C01826=1220.684,210.182,-57.626,-177.358,6.193,148.333
C01827=1220.680,210.431,-57.649,-177.356,6.195,148.332
C01828=1220.676,210.681,-57.674,-177.353,6.197,148.332
C01829=1220.671,210.929,-57.699,-177.350,6.199,148.332
C01830=1220.666,211.199,-57.725,-177.347,6.200,148.331
C01831=1220.661,211.469,-57.751,-177.345,6.202,148.331
C01832=1220.656,211.739,-57.778,-177.342,6.204,148.330
C01833=1220.651,212.011,-57.804,-177.339,6.206,148.330
C01834=1220.647,212.259,-57.829,-177.337,6.208,148.330
C01835=1220.642,212.508,-57.853,-177.334,6.209,148.329
C01836=1220.637,212.757,-57.877,-177.331,6.211,148.329
C01837=1220.633,213.006,-57.902,-177.329,6.213,148.329
C01838=1220.628,213.254,-57.926,-177.326,6.215,148.328
C01839=1220.623,213.503,-57.951,-177.323,6.217,148.328
C01840=1220.620,213.752,-57.975,-177.321,6.219,148.328
C01841=1220.614,214.001,-58.000,-177.318,6.220,148.328
C01842=1220.610,214.249,-58.024,-177.316,6.222,148.327
C01843=1220.606,214.498,-58.050,-177.313,6.224,148.327
C01844=1220.601,214.747,-58.074,-177.311,6.225,148.326
C01845=1220.596,214.995,-58.099,-177.308,6.227,148.326
C01846=1220.592,215.244,-58.123,-177.306,6.229,148.326
C01847=1220.587,215.493,-58.148,-177.303,6.231,148.325
C01848=1220.583,215.742,-58.172,-177.300,6.233,148.325
C01849=1220.578,215.991,-58.197,-177.298,6.234,148.325
C01850=1220.574,216.239,-58.221,-177.295,6.236,148.324
C01851=1220.569,216.487,-58.246,-177.292,6.238,148.324
C01852=1220.565,216.737,-58.271,-177.290,6.240,148.324
C01853=1220.560,216.985,-58.295,-177.287,6.242,148.323
C01854=1220.556,217.235,-58.321,-177.285,6.244,148.323
C01855=1220.551,217.483,-58.345,-177.282,6.246,148.323
C01856=1220.546,217.732,-58.369,-177.279,6.247,148.322
C01857=1220.543,217.980,-58.394,-177.277,6.250,148.322
C01858=1220.538,218.229,-58.419,-177.274,6.251,148.322
C01859=1220.532,218.478,-58.444,-177.272,6.252,148.322
C01860=1220.529,218.727,-58.468,-177.270,6.254,148.321
C01861=1220.524,218.975,-58.494,-177.267,6.256,148.321
C01862=1220.520,219.224,-58.518,-177.265,6.258,148.321
C01863=1220.515,219.473,-58.543,-177.262,6.260,148.320
C01864=1220.511,219.722,-58.568,-177.259,6.262,148.320
C01865=1220.506,219.970,-58.593,-177.257,6.264,148.320
C01866=1220.501,220.219,-58.617,-177.254,6.265,148.319
C01867=1220.497,220.468,-58.643,-177.251,6.267,148.319
C01868=1220.493,220.716,-58.667,-177.249,6.269,148.319
C01869=1220.488,220.965,-58.692,-177.246,6.271,148.318
C01870=1220.483,221.214,-58.717,-177.243,6.273,148.318
C01871=1220.479,221.463,-58.742,-177.241,6.275,148.318
C01872=1220.474,221.711,-58.767,-177.238,6.277,148.317
C01873=1220.470,221.960,-58.792,-177.236,6.279,148.317
C01874=1220.465,222.209,-58.817,-177.233,6.281,148.317
C01875=1220.461,222.457,-58.842,-177.231,6.282,148.317
C01876=1220.456,222.706,-58.867,-177.228,6.284,148.316
C01877=1220.451,222.955,-58.891,-177.226,6.286,148.316
C01878=1220.447,223.204,-58.917,-177.223,6.287,148.316
C01879=1220.443,223.452,-58.941,-177.221,6.289,148.315
C01880=1220.438,223.701,-58.967,-177.218,6.291,148.315
C01881=1220.433,223.950,-58.992,-177.216,6.293,148.315
C01882=1220.429,224.198,-59.017,-177.213,6.295,148.314
C01883=1220.425,224.447,-59.042,-177.210,6.297,148.314
C01884=1220.420,224.696,-59.067,-177.208,6.299,148.314
C01885=1220.415,224.944,-59.092,-177.206,6.301,148.314
C01886=1220.411,225.193,-59.118,-177.203,6.302,148.313
C01887=1220.406,225.442,-59.142,-177.200,6.304,148.313
C01888=1220.402,225.691,-59.168,-177.198,6.306,148.313
C01889=1220.398,225.939,-59.193,-177.195,6.308,148.312
C01890=1220.393,226.188,-59.218,-177.192,6.310,148.312
C01891=1220.389,226.437,-59.244,-177.190,6.312,148.312
C01892=1220.384,226.685,-59.268,-177.187,6.314,148.311
C01893=1220.379,226.934,-59.294,-177.185,6.316,148.311
C01894=1220.375,227.182,-59.320,-177.182,6.318,148.311
C01895=1220.370,227.432,-59.345,-177.180,6.319,148.311
C01896=1220.366,227.680,-59.369,-177.177,6.321,148.310
C01897=1220.362,227.928,-59.395,-177.174,6.323,148.310
C01898=1220.357,228.177,-59.420,-177.172,6.325,148.310
C01899=1220.352,228.426,-59.446,-177.169,6.327,148.309
C01900=1220.348,228.675,-59.471,-177.167,6.329,148.309
C01901=1220.343,228.923,-59.496,-177.164,6.331,148.309
C01902=1220.339,229.172,-59.522,-177.162,6.333,148.309
C01903=1220.334,229.420,-59.547,-177.159,6.335,148.308
C01904=1220.329,229.670,-59.572,-177.157,6.337,148.308
C01905=1220.325,229.919,-59.598,-177.154,6.338,148.308
C01906=1220.320,230.167,-59.623,-177.151,6.340,148.307
C01907=1220.316,230.415,-59.649,-177.149,6.342,148.307
C01908=1220.311,230.664,-59.674,-177.147,6.344,148.307
C01909=1220.307,230.913,-59.699,-177.144,6.346,148.306
C01910=1220.303,231.162,-59.725,-177.141,6.348,148.306
C01911=1220.298,231.410,-59.751,-177.139,6.350,148.306
C01912=1220.294,231.659,-59.776,-177.136,6.352,148.306
C01913=1220.289,231.907,-59.802,-177.133,6.354,148.305
C01914=1220.284,232.156,-59.827,-177.131,6.356,148.305
C01915=1220.280,232.405,-59.852,-177.129,6.358,148.305
C01916=1220.276,232.654,-59.878,-177.126,6.360,148.304
C01917=1220.271,232.902,-59.904,-177.123,6.361,148.304
C01918=1220.267,233.151,-59.929,-177.121,6.363,148.304
C01919=1220.262,233.400,-59.955,-177.118,6.365,148.303
C01920=1220.258,233.648,-59.980,-177.116,6.367,148.303
C01921=1220.253,233.896,-60.006,-177.113,6.369,148.303
C01922=1220.249,234.145,-60.032,-177.111,6.371,148.303
C01923=1220.244,234.393,-60.057,-177.108,6.373,148.302
C01924=1220.240,234.643,-60.082,-177.106,6.375,148.302
C01925=1220.236,234.892,-60.108,-177.103,6.377,148.302
C01926=1220.231,235.140,-60.134,-177.101,6.379,148.302
C01927=1220.227,235.388,-60.159,-177.098,6.381,148.301
C01928=1220.222,235.638,-60.186,-177.096,6.383,148.301
C01929=1220.217,235.886,-60.211,-177.093,6.384,148.301
C01930=1220.213,236.135,-60.237,-177.091,6.387,148.301
C01931=1220.208,236.383,-60.263,-177.088,6.388,148.300
C01932=1220.204,236.631,-60.289,-177.086,6.390,148.300
C01933=1220.200,236.880,-60.314,-177.083,6.392,148.300
C01934=1220.195,237.151,-60.342,-177.080,6.394,148.299
C01935=1220.190,237.423,-60.370,-177.077,6.397,148.299
C01936=1220.185,237.694,-60.399,-177.074,6.399,148.299
C01937=1220.180,237.966,-60.427,-177.072,6.400,148.298
C01938=1220.175,238.214,-60.453,-177.070,6.403,148.298
C01939=1220.171,238.463,-60.479,-177.067,6.405,148.298
C01940=1220.167,238.712,-60.504,-177.064,6.406,148.298
C01941=1220.162,238.961,-60.530,-177.062,6.408,148.297
C01942=1220.157,239.208,-60.557,-177.059,6.410,148.297
C01943=1220.153,239.457,-60.583,-177.057,6.412,148.297
C01944=1220.149,239.706,-60.608,-177.054,6.414,148.297
C01945=1220.144,239.955,-60.634,-177.051,6.417,148.296
C01946=1220.139,240.204,-60.660,-177.049,6.419,148.296
C01947=1220.135,240.452,-60.687,-177.047,6.421,148.296
C01948=1220.131,240.700,-60.712,-177.044,6.423,148.296
C01949=1220.126,240.949,-60.738,-177.041,6.425,148.295
C01950=1220.121,241.198,-60.764,-177.039,6.427,148.295
C01951=1220.118,241.446,-60.791,-177.036,6.428,148.295
C01952=1220.113,241.695,-60.816,-177.034,6.431,148.295
C01953=1220.108,241.944,-60.843,-177.031,6.432,148.294
C01954=1220.104,242.192,-60.868,-177.029,6.434,148.294
C01955=1220.100,242.441,-60.895,-177.026,6.436,148.294
C01956=1220.095,242.689,-60.921,-177.024,6.438,148.294
C01957=1220.090,242.939,-60.947,-177.021,6.440,148.293
C01958=1220.086,243.186,-60.973,-177.019,6.442,148.293
C01959=1220.081,243.435,-60.999,-177.016,6.444,148.293
C01960=1220.077,243.684,-61.025,-177.014,6.446,148.293
C01961=1220.073,243.932,-61.052,-177.011,6.448,148.292
C01962=1220.068,244.181,-61.078,-177.009,6.450,148.292
C01963=1220.064,244.429,-61.104,-177.006,6.453,148.292
C01964=1220.060,244.678,-61.130,-177.003,6.455,148.292
C01965=1220.054,244.927,-61.156,-177.001,6.457,148.291
C01966=1220.050,245.175,-61.183,-176.998,6.459,148.291
C01967=1220.045,245.424,-61.209,-176.996,6.461,148.291
C01968=1220.041,245.672,-61.235,-176.993,6.463,148.291
C01969=1220.037,245.921,-61.261,-176.991,6.464,148.290
C01970=1220.032,246.169,-61.288,-176.988,6.466,148.290
C01971=1220.028,246.418,-61.314,-176.986,6.469,148.290
C01972=1220.024,246.667,-61.341,-176.983,6.470,148.290
C01973=1220.019,246.916,-61.367,-176.981,6.472,148.289
C01974=1220.014,247.163,-61.393,-176.979,6.474,148.289
C01975=1220.010,247.412,-61.419,-176.976,6.476,148.289
C01976=1220.005,247.661,-61.446,-176.973,6.479,148.289
C01977=1220.001,247.909,-61.472,-176.970,6.481,148.288
C01978=1219.997,248.158,-61.498,-176.968,6.483,148.288
C01979=1219.992,248.407,-61.525,-176.966,6.485,148.288
C01980=1219.988,248.655,-61.551,-176.963,6.487,148.288
C01981=1219.984,248.903,-61.578,-176.961,6.489,148.287
C01982=1219.979,249.153,-61.605,-176.958,6.491,148.287
C01983=1219.975,249.401,-61.631,-176.956,6.493,148.287
C01984=1219.970,249.650,-61.657,-176.953,6.495,148.287
C01985=1219.966,249.898,-61.684,-176.951,6.497,148.286
C01986=1219.961,250.147,-61.711,-176.948,6.500,148.286
C01987=1219.957,250.395,-61.737,-176.945,6.501,148.286
C01988=1219.952,250.644,-61.764,-176.943,6.504,148.286
C01989=1219.948,250.892,-61.790,-176.940,6.506,148.285
C01990=1219.943,251.141,-61.817,-176.938,6.507,148.285
C01991=1219.939,251.390,-61.844,-176.935,6.510,148.285
C01992=1219.935,251.638,-61.870,-176.933,6.511,148.285
C01993=1219.930,251.886,-61.897,-176.930,6.513,148.284
C01994=1219.926,252.135,-61.923,-176.928,6.516,148.284
C01995=1219.921,252.384,-61.950,-176.925,6.518,148.284
C01996=1219.917,252.632,-61.977,-176.922,6.520,148.284
C01997=1219.913,252.880,-62.004,-176.920,6.522,148.284
C01998=1219.908,253.129,-62.030,-176.918,6.524,148.283
C01999=1219.904,253.378,-62.056,-176.915,6.526,148.283
C02000=1219.899,253.626,-62.083,-176.913,6.528,148.283
C02001=1219.894,253.875,-62.111,-176.910,6.530,148.283
C02002=1219.891,254.123,-62.137,-176.908,6.532,148.282
C02003=1219.886,254.372,-62.163,-176.905,6.535,148.282
C02004=1219.881,254.620,-62.190,-176.902,6.537,148.282
C02005=1219.877,254.869,-62.217,-176.900,6.539,148.282
C02006=1219.872,255.117,-62.244,-176.898,6.541,148.282
C02007=1219.868,255.366,-62.271,-176.895,6.543,148.281
C02008=1219.863,255.614,-62.298,-176.893,6.545,148.281
C02009=1219.859,255.862,-62.325,-176.890,6.547,148.281
C02010=1219.854,256.111,-62.352,-176.888,6.549,148.281
C02011=1219.850,256.359,-62.379,-176.885,6.552,148.281
C02012=1219.846,256.609,-62.405,-176.882,6.554,148.280
C02013=1219.841,256.857,-62.432,-176.880,6.556,148.280
C02014=1219.837,257.106,-62.459,-176.878,6.558,148.280
C02015=1219.832,257.354,-62.486,-176.875,6.560,148.280
C02016=1219.828,257.603,-62.513,-176.873,6.562,148.280
C02017=1219.824,257.851,-62.539,-176.870,6.565,148.279
C02018=1219.819,258.099,-62.567,-176.867,6.566,148.279
C02019=1219.814,258.348,-62.594,-176.865,6.569,148.279
C02020=1219.810,258.596,-62.621,-176.862,6.570,148.279
C02021=1219.806,258.846,-62.648,-176.860,6.572,148.278
C02022=1219.802,259.093,-62.675,-176.858,6.575,148.278
C02023=1219.797,259.342,-62.702,-176.855,6.576,148.278
C02024=1219.793,259.590,-62.729,-176.852,6.579,148.278
C02025=1219.788,259.839,-62.756,-176.850,6.581,148.278
C02026=1219.783,260.087,-62.783,-176.847,6.583,148.277
C02027=1219.779,260.336,-62.811,-176.845,6.585,148.277
C02028=1219.775,260.585,-62.837,-176.842,6.587,148.277
C02029=1219.771,260.833,-62.864,-176.840,6.589,148.277
C02030=1219.766,261.081,-62.892,-176.837,6.592,148.277
C02031=1219.762,261.329,-62.919,-176.835,6.594,148.276
C02032=1219.757,261.578,-62.946,-176.832,6.596,148.276
C02033=1219.752,261.826,-62.973,-176.830,6.598,148.276
C02034=1219.748,262.076,-63.001,-176.828,6.600,148.276
C02035=1219.744,262.324,-63.028,-176.824,6.603,148.275
C02036=1219.739,262.572,-63.056,-176.822,6.605,148.275
C02037=1219.735,262.820,-63.082,-176.820,6.607,148.275
C02038=1219.730,263.093,-63.112,-176.817,6.609,148.275
C02039=1219.725,263.366,-63.141,-176.814,6.612,148.275
C02040=1219.721,263.639,-63.172,-176.812,6.614,148.274
C02041=1219.716,263.911,-63.202,-176.809,6.617,148.274
C02042=1219.711,264.160,-63.229,-176.806,6.619,148.274
C02043=1219.707,264.408,-63.257,-176.804,6.621,148.274
C02044=1219.702,264.656,-63.284,-176.801,6.623,148.274
C02045=1219.698,264.905,-63.311,-176.799,6.626,148.273
C02046=1219.694,265.153,-63.339,-176.796,6.628,148.273
C02047=1219.689,265.402,-63.366,-176.794,6.630,148.273
C02048=1219.685,265.650,-63.393,-176.791,6.632,148.273
C02049=1219.681,265.899,-63.421,-176.789,6.634,148.273
C02050=1219.676,266.147,-63.448,-176.786,6.637,148.272
C02051=1219.672,266.395,-63.476,-176.784,6.639,148.272
C02052=1219.667,266.644,-63.503,-176.781,6.641,148.272
C02053=1219.663,266.893,-63.531,-176.779,6.643,148.272
C02054=1219.658,267.141,-63.559,-176.776,6.645,148.272
C02055=1219.654,267.390,-63.586,-176.774,6.648,148.272
C02056=1219.650,267.638,-63.614,-176.771,6.650,148.271
C02057=1219.645,267.887,-63.641,-176.769,6.652,148.271
C02058=1219.641,268.134,-63.669,-176.766,6.654,148.271
C02059=1219.636,268.383,-63.696,-176.763,6.656,148.271
C02060=1219.632,268.632,-63.724,-176.761,6.659,148.271
C02061=1219.628,268.880,-63.751,-176.759,6.660,148.270
C02062=1219.623,269.128,-63.779,-176.756,6.663,148.270
C02063=1219.619,269.377,-63.806,-176.753,6.665,148.270
C02064=1219.614,269.625,-63.835,-176.751,6.668,148.270
C02065=1219.610,269.874,-63.862,-176.749,6.669,148.270
C02066=1219.606,270.122,-63.890,-176.746,6.672,148.270
C02067=1219.601,270.371,-63.917,-176.744,6.674,148.269
C02068=1219.597,270.619,-63.945,-176.741,6.677,148.269
C02069=1219.593,270.867,-63.973,-176.738,6.678,148.269
C02070=1219.588,271.116,-64.001,-176.736,6.681,148.269
C02071=1219.583,271.364,-64.028,-176.734,6.683,148.269
C02072=1219.579,271.613,-64.056,-176.731,6.686,148.269
C02073=1219.575,271.861,-64.084,-176.729,6.688,148.269
C02074=1219.571,272.110,-64.112,-176.726,6.690,148.268
C02075=1219.566,272.358,-64.139,-176.724,6.692,148.268
C02076=1219.561,272.606,-64.167,-176.721,6.695,148.268
C02077=1219.558,272.855,-64.195,-176.719,6.697,148.268
C02078=1219.553,273.103,-64.222,-176.716,6.699,148.268
C02079=1219.548,273.352,-64.251,-176.714,6.701,148.267
C02080=1219.544,273.600,-64.279,-176.711,6.704,148.267
C02081=1219.540,273.848,-64.307,-176.709,6.706,148.267
C02082=1219.536,274.097,-64.334,-176.706,6.708,148.267
C02083=1219.531,274.345,-64.362,-176.704,6.710,148.267
C02084=1219.526,274.593,-64.390,-176.701,6.713,148.267
C02085=1219.523,274.842,-64.418,-176.699,6.715,148.266
C02086=1219.518,275.090,-64.445,-176.697,6.717,148.266
C02087=1219.513,275.339,-64.474,-176.694,6.719,148.266
C02088=1219.509,275.587,-64.502,-176.692,6.722,148.266
C02089=1219.505,275.836,-64.530,-176.689,6.724,148.266
C02090=1219.500,276.084,-64.559,-176.687,6.726,148.266
C02091=1219.496,276.332,-64.587,-176.684,6.729,148.265
C02092=1219.492,276.581,-64.614,-176.682,6.731,148.265
C02093=1219.487,276.829,-64.642,-176.679,6.733,148.265
C02094=1219.483,277.078,-64.670,-176.677,6.735,148.265
C02095=1219.479,277.326,-64.698,-176.674,6.738,148.265
C02096=1219.474,277.575,-64.727,-176.672,6.740,148.265
C02097=1219.470,277.822,-64.755,-176.669,6.742,148.265
C02098=1219.465,278.071,-64.783,-176.667,6.744,148.264
C02099=1219.461,278.319,-64.811,-176.664,6.747,148.264
C02100=1219.457,278.568,-64.839,-176.662,6.749,148.264
C02101=1219.452,278.816,-64.868,-176.659,6.751,148.264
C02102=1219.448,279.064,-64.896,-176.657,6.754,148.264
C02103=1219.443,279.313,-64.924,-176.654,6.756,148.264
C02104=1219.440,279.561,-64.952,-176.652,6.758,148.264
C02105=1219.435,279.809,-64.980,-176.650,6.760,148.263
C02106=1219.431,280.058,-65.009,-176.647,6.763,148.263
C02107=1219.426,280.306,-65.036,-176.645,6.765,148.263
C02108=1219.422,280.555,-65.065,-176.642,6.767,148.263
C02109=1219.418,280.803,-65.093,-176.639,6.770,148.263
C02110=1219.413,281.052,-65.122,-176.637,6.773,148.263
C02111=1219.409,281.299,-65.150,-176.635,6.774,148.262
C02112=1219.404,281.548,-65.178,-176.632,6.777,148.262
C02113=1219.400,281.797,-65.206,-176.630,6.780,148.262
C02114=1219.395,282.045,-65.235,-176.627,6.782,148.262
C02115=1219.392,282.293,-65.264,-176.625,6.784,148.262
C02116=1219.387,282.541,-65.292,-176.622,6.787,148.262
C02117=1219.383,282.790,-65.320,-176.620,6.789,148.262
C02118=1219.378,283.038,-65.349,-176.618,6.791,148.262
C02119=1219.374,283.287,-65.377,-176.615,6.794,148.262
C02120=1219.370,283.535,-65.405,-176.612,6.796,148.261
C02121=1219.365,283.783,-65.434,-176.610,6.798,148.261
C02122=1219.361,284.032,-65.463,-176.608,6.801,148.261
C02123=1219.356,284.280,-65.491,-176.605,6.803,148.261
C02124=1219.352,284.528,-65.519,-176.603,6.805,148.261
C02125=1219.347,284.777,-65.548,-176.600,6.808,148.261
C02126=1219.343,285.025,-65.577,-176.598,6.810,148.261
C02127=1219.339,285.273,-65.605,-176.595,6.812,148.261
C02128=1219.334,285.522,-65.633,-176.593,6.815,148.260
C02129=1219.331,285.770,-65.662,-176.590,6.817,148.260
C02130=1219.326,286.018,-65.691,-176.588,6.819,148.260
C02131=1219.321,286.267,-65.719,-176.585,6.822,148.260
C02132=1219.318,286.515,-65.748,-176.583,6.824,148.260
C02133=1219.313,286.763,-65.777,-176.581,6.827,148.260
C02134=1219.308,287.012,-65.805,-176.578,6.830,148.260
C02135=1219.305,287.260,-65.834,-176.575,6.831,148.259
C02136=1219.300,287.508,-65.863,-176.573,6.834,148.259
C02137=1219.295,287.757,-65.891,-176.571,6.837,148.259
C02138=1219.292,288.005,-65.920,-176.569,6.839,148.259
C02139=1219.287,288.253,-65.949,-176.566,6.841,148.259
C02140=1219.282,288.501,-65.978,-176.563,6.844,148.259
C02141=1219.278,288.750,-66.007,-176.561,6.846,148.259
C02142=1219.273,289.024,-66.038,-176.558,6.849,148.259
C02143=1219.268,289.299,-66.070,-176.556,6.851,148.259
C02144=1219.263,289.572,-66.102,-176.553,6.854,148.259
C02145=1219.258,289.846,-66.134,-176.550,6.857,148.258
C02146=1219.255,290.095,-66.162,-176.548,6.859,148.258
C02147=1219.251,290.343,-66.191,-176.546,6.861,148.258
C02148=1219.246,290.592,-66.220,-176.543,6.864,148.258
C02149=1219.241,290.839,-66.249,-176.541,6.866,148.258
C02150=1219.238,291.087,-66.278,-176.538,6.868,148.258
C02151=1219.233,291.336,-66.307,-176.536,6.871,148.258
C02152=1219.229,291.584,-66.336,-176.533,6.873,148.258
C02153=1219.224,291.833,-66.365,-176.531,6.875,148.258
C02154=1219.220,292.081,-66.394,-176.528,6.879,148.258
C02155=1219.215,292.330,-66.423,-176.526,6.881,148.257
C02156=1219.211,292.577,-66.451,-176.524,6.884,148.257
C02157=1219.207,292.825,-66.481,-176.521,6.886,148.257
C02158=1219.203,293.074,-66.509,-176.519,6.888,148.257
C02159=1219.199,293.322,-66.539,-176.516,6.891,148.257
C02160=1219.194,293.570,-66.568,-176.514,6.893,148.257
C02161=1219.189,293.819,-66.597,-176.511,6.895,148.257
C02162=1219.185,294.067,-66.626,-176.509,6.898,148.257
C02163=1219.182,294.315,-66.655,-176.507,6.900,148.257
C02164=1219.177,294.564,-66.684,-176.505,6.902,148.257
C02165=1219.172,294.812,-66.713,-176.502,6.906,148.257
C02166=1219.168,295.060,-66.742,-176.500,6.908,148.257
C02167=1219.164,295.308,-66.772,-176.497,6.910,148.256
C02168=1219.159,295.557,-66.801,-176.495,6.913,148.256
C02169=1219.155,295.805,-66.830,-176.492,6.915,148.256
C02170=1219.151,296.053,-66.859,-176.490,6.918,148.256
C02171=1219.146,296.301,-66.888,-176.488,6.920,148.256
C02172=1219.142,296.549,-66.918,-176.485,6.922,148.256
C02173=1219.138,296.798,-66.947,-176.482,6.925,148.256
C02174=1219.133,297.047,-66.976,-176.480,6.927,148.256
C02175=1219.129,297.295,-67.006,-176.478,6.930,148.256
C02176=1219.125,297.542,-67.035,-176.475,6.933,148.256
C02177=1219.120,297.791,-67.064,-176.473,6.935,148.256
C02178=1219.116,298.039,-67.094,-176.471,6.938,148.256
C02179=1219.112,298.288,-67.122,-176.468,6.940,148.255
C02180=1219.108,298.536,-67.152,-176.465,6.943,148.255
C02181=1219.103,298.784,-67.181,-176.463,6.945,148.255
C02182=1219.099,299.032,-67.210,-176.461,6.947,148.255
C02183=1219.094,299.280,-67.240,-176.458,6.950,148.255
C02184=1219.090,299.528,-67.269,-176.456,6.952,148.255
C02185=1219.086,299.777,-67.299,-176.454,6.955,148.255
C02186=1219.082,300.025,-67.328,-176.452,6.958,148.255
C02187=1219.078,300.273,-67.358,-176.449,6.960,148.255
C02188=1219.073,300.522,-67.387,-176.446,6.963,148.255
C02189=1219.069,300.770,-67.416,-176.444,6.965,148.255
C02190=1219.065,301.018,-67.446,-176.442,6.967,148.255
C02191=1219.060,301.266,-67.475,-176.439,6.970,148.255
C02192=1219.056,301.514,-67.504,-176.437,6.972,148.255
C02193=1219.052,301.762,-67.534,-176.435,6.975,148.255
C02194=1219.047,302.011,-67.564,-176.433,6.977,148.254
C02195=1219.043,302.259,-67.593,-176.430,6.981,148.254
C02196=1219.039,302.507,-67.623,-176.428,6.983,148.254
C02197=1219.034,302.756,-67.652,-176.426,6.985,148.254
C02198=1219.030,303.004,-67.682,-176.423,6.988,148.254
C02199=1219.026,303.251,-67.712,-176.421,6.990,148.254
C02200=1219.022,303.500,-67.741,-176.418,6.993,148.254
C02201=1219.017,303.748,-67.771,-176.416,6.995,148.254
C02202=1219.013,303.997,-67.801,-176.414,6.998,148.254
C02203=1219.009,304.245,-67.830,-176.411,7.000,148.254
C02204=1219.005,304.493,-67.860,-176.409,7.003,148.254
C02205=1219.001,304.741,-67.890,-176.406,7.006,148.254
C02206=1218.996,304.989,-67.920,-176.404,7.008,148.254
C02207=1218.992,305.238,-67.950,-176.402,7.010,148.254
C02208=1218.988,305.486,-67.979,-176.399,7.013,148.254
C02209=1218.983,305.734,-68.008,-176.397,7.015,148.254
C02210=1218.979,305.982,-68.039,-176.394,7.018,148.254
C02211=1218.974,306.230,-68.068,-176.392,7.021,148.254
C02212=1218.970,306.478,-68.098,-176.390,7.024,148.254
C02213=1218.966,306.726,-68.127,-176.387,7.026,148.254
C02214=1218.962,306.975,-68.158,-176.385,7.028,148.254
C02215=1218.957,307.223,-68.188,-176.383,7.031,148.254
C02216=1218.953,307.471,-68.217,-176.381,7.033,148.253
C02217=1218.949,307.719,-68.248,-176.378,7.036,148.253
C02218=1218.945,307.968,-68.277,-176.376,7.039,148.253
C02219=1218.940,308.216,-68.307,-176.374,7.041,148.254
C02220=1218.936,308.464,-68.338,-176.371,7.044,148.254
C02221=1218.932,308.712,-68.367,-176.369,7.046,148.254
C02222=1218.927,308.960,-68.397,-176.367,7.049,148.253
C02223=1218.923,309.208,-68.427,-176.365,7.052,148.253
C02224=1218.919,309.457,-68.457,-176.362,7.055,148.253
C02225=1218.915,309.704,-68.487,-176.360,7.057,148.253
C02226=1218.910,309.953,-68.517,-176.358,7.059,148.253
C02227=1218.906,310.200,-68.547,-176.355,7.062,148.253
C02228=1218.902,310.449,-68.577,-176.353,7.064,148.253
C02229=1218.897,310.697,-68.607,-176.350,7.067,148.253
C02230=1218.893,310.945,-68.637,-176.348,7.070,148.253
C02231=1218.888,311.194,-68.667,-176.345,7.073,148.253
C02232=1218.884,311.441,-68.697,-176.343,7.075,148.253
C02233=1218.881,311.690,-68.728,-176.341,7.077,148.253
C02234=1218.876,311.938,-68.758,-176.339,7.080,148.253
C02235=1218.872,312.186,-68.788,-176.337,7.083,148.253
C02236=1218.867,312.434,-68.818,-176.334,7.086,148.253
C02237=1218.863,312.682,-68.848,-176.332,7.088,148.253
C02238=1218.858,312.931,-68.878,-176.329,7.091,148.253
C02239=1218.854,313.178,-68.908,-176.327,7.093,148.253
C02240=1218.850,313.427,-68.938,-176.325,7.096,148.253
C02241=1218.846,313.674,-68.968,-176.323,7.098,148.253
C02242=1218.842,313.923,-69.000,-176.321,7.101,148.253
C02243=1218.837,314.171,-69.029,-176.318,7.104,148.253
C02244=1218.833,314.419,-69.060,-176.316,7.106,148.253
C02245=1218.829,314.667,-69.090,-176.313,7.109,148.253
C02246=1218.824,314.943,-69.124,-176.311,7.112,148.253
C02247=1218.820,315.219,-69.157,-176.309,7.115,148.253
C02248=1218.815,315.495,-69.191,-176.306,7.118,148.253
C02249=1218.810,315.771,-69.225,-176.303,7.121,148.253
C02250=1218.806,316.019,-69.255,-176.302,7.123,148.253
C02251=1218.801,316.267,-69.285,-176.299,7.126,148.253
C02252=1218.797,316.515,-69.315,-176.297,7.128,148.253
C02253=1218.793,316.763,-69.346,-176.294,7.131,148.253
C02254=1218.788,317.012,-69.377,-176.292,7.134,148.253
C02255=1218.785,317.260,-69.407,-176.290,7.137,148.253
C02256=1218.780,317.508,-69.438,-176.288,7.139,148.253
C02257=1218.776,317.755,-69.468,-176.285,7.142,148.253
C02258=1218.771,318.003,-69.498,-176.283,7.144,148.253
C02259=1218.767,318.253,-69.529,-176.280,7.148,148.253
C02260=1218.763,318.500,-69.559,-176.279,7.150,148.254
C02261=1218.759,318.748,-69.590,-176.277,7.152,148.253
C02262=1218.754,318.996,-69.621,-176.274,7.155,148.253
C02263=1218.751,319.245,-69.651,-176.272,7.158,148.253
C02264=1218.746,319.493,-69.682,-176.270,7.161,148.254
C02265=1218.742,319.740,-69.712,-176.268,7.163,148.254
C02266=1218.738,319.988,-69.743,-176.265,7.166,148.254
C02267=1218.734,320.237,-69.774,-176.263,7.168,148.254
C02268=1218.729,320.485,-69.803,-176.261,7.172,148.254
C02269=1218.725,320.733,-69.834,-176.259,7.174,148.254
C02270=1218.720,320.981,-69.865,-176.256,7.176,148.254
C02271=1218.716,321.230,-69.896,-176.254,7.180,148.254
C02272=1218.712,321.477,-69.926,-176.252,7.182,148.254
C02273=1218.708,321.725,-69.957,-176.249,7.185,148.254
C02274=1218.703,321.973,-69.988,-176.248,7.187,148.254
C02275=1218.700,322.222,-70.018,-176.245,7.190,148.254
C02276=1218.695,322.470,-70.049,-176.243,7.193,148.254
C02277=1218.691,322.717,-70.080,-176.240,7.196,148.254
C02278=1218.687,322.966,-70.111,-176.239,7.198,148.254
C02279=1218.683,323.214,-70.141,-176.237,7.200,148.254
C02280=1218.678,323.461,-70.173,-176.234,7.204,148.254
C02281=1218.674,323.710,-70.204,-176.232,7.206,148.254
C02282=1218.670,323.958,-70.234,-176.230,7.209,148.254
C02283=1218.665,324.206,-70.265,-176.228,7.211,148.254
C02284=1218.662,324.454,-70.296,-176.225,7.215,148.254
C02285=1218.657,324.702,-70.327,-176.223,7.217,148.254
C02286=1218.653,324.950,-70.357,-176.221,7.220,148.255
C02287=1218.649,325.199,-70.388,-176.219,7.222,148.255
C02288=1218.644,325.446,-70.420,-176.216,7.225,148.255
C02289=1218.640,325.694,-70.450,-176.215,7.228,148.255
C02290=1218.636,325.942,-70.481,-176.213,7.230,148.255
C02291=1218.632,326.190,-70.512,-176.210,7.233,148.255
C02292=1218.627,326.438,-70.543,-176.208,7.236,148.255
C02293=1218.624,326.686,-70.575,-176.206,7.239,148.255
C02294=1218.619,326.934,-70.605,-176.204,7.241,148.255
C02295=1218.615,327.183,-70.636,-176.201,7.244,148.255
C02296=1218.611,327.430,-70.667,-176.200,7.247,148.255
C02297=1218.606,327.678,-70.697,-176.197,7.250,148.255
C02298=1218.603,327.926,-70.729,-176.195,7.252,148.255
C02299=1218.598,328.174,-70.760,-176.193,7.255,148.255
C02300=1218.593,328.422,-70.791,-176.191,7.258,148.256
C02301=1218.590,328.670,-70.823,-176.189,7.260,148.256
C02302=1218.585,328.918,-70.853,-176.186,7.263,148.256
C02303=1218.581,329.167,-70.885,-176.185,7.266,148.256
C02304=1218.577,329.414,-70.916,-176.182,7.269,148.256
C02305=1218.573,329.663,-70.947,-176.180,7.271,148.256
C02306=1218.568,329.911,-70.978,-176.178,7.274,148.256
C02307=1218.564,330.158,-71.009,-176.176,7.277,148.256
C02308=1218.560,330.407,-71.041,-176.173,7.280,148.256
C02309=1218.556,330.654,-71.072,-176.172,7.282,148.256
C02310=1218.552,330.903,-71.103,-176.170,7.285,148.256
C02311=1218.547,331.151,-71.134,-176.167,7.288,148.256
C02312=1218.543,331.399,-71.166,-176.166,7.291,148.257
C02313=1218.539,331.647,-71.197,-176.163,7.294,148.257
C02314=1218.534,331.894,-71.228,-176.161,7.296,148.257
C02315=1218.530,332.143,-71.259,-176.159,7.299,148.257
C02316=1218.526,332.390,-71.291,-176.157,7.302,148.257
C02317=1218.522,332.639,-71.322,-176.155,7.305,148.257
C02318=1218.518,332.886,-71.353,-176.153,7.307,148.257
C02319=1218.514,333.135,-71.384,-176.150,7.310,148.257
C02320=1218.509,333.382,-71.416,-176.149,7.313,148.257
C02321=1218.505,333.631,-71.447,-176.147,7.315,148.258
C02322=1218.501,333.878,-71.478,-176.144,7.318,148.258
C02323=1218.497,334.127,-71.510,-176.143,7.321,148.258
C02324=1218.493,334.374,-71.541,-176.140,7.324,148.258
C02325=1218.488,334.623,-71.573,-176.138,7.327,148.258
C02326=1218.484,334.871,-71.604,-176.136,7.330,148.258
C02327=1218.480,335.119,-71.636,-176.134,7.332,148.258
C02328=1218.475,335.367,-71.667,-176.132,7.335,148.258
C02329=1218.472,335.615,-71.699,-176.130,7.338,148.258
C02330=1218.467,335.862,-71.730,-176.128,7.340,148.258
C02331=1218.463,336.111,-71.761,-176.126,7.344,148.259
C02332=1218.459,336.358,-71.793,-176.124,7.346,148.259
C02333=1218.455,336.606,-71.825,-176.122,7.349,148.259
C02334=1218.451,336.855,-71.856,-176.120,7.352,148.259
C02335=1218.446,337.102,-71.888,-176.118,7.355,148.259
C02336=1218.443,337.350,-71.920,-176.116,7.357,148.259
C02337=1218.438,337.598,-71.950,-176.114,7.360,148.259
C02338=1218.433,337.847,-71.983,-176.112,7.363,148.260
C02339=1218.429,338.094,-72.014,-176.110,7.365,148.260
C02340=1218.425,338.342,-72.046,-176.108,7.369,148.260
C02341=1218.421,338.591,-72.077,-176.106,7.371,148.260
C02342=1218.417,338.838,-72.109,-176.103,7.374,148.260
C02343=1218.413,339.086,-72.141,-176.102,7.377,148.260
C02344=1218.408,339.334,-72.173,-176.100,7.379,148.260
C02345=1218.405,339.582,-72.205,-176.098,7.383,148.261
C02346=1218.400,339.830,-72.235,-176.096,7.385,148.261
C02347=1218.396,340.078,-72.268,-176.093,7.388,148.261
C02348=1218.392,340.326,-72.300,-176.092,7.391,148.261
C02349=1218.388,340.573,-72.331,-176.090,7.394,148.261
C02350=1218.383,340.851,-72.367,-176.088,7.396,148.261
C02351=1218.378,341.129,-72.402,-176.085,7.400,148.261
C02352=1218.374,341.407,-72.438,-176.083,7.403,148.262
C02353=1218.369,341.685,-72.474,-176.081,7.406,148.262
C02354=1218.365,341.933,-72.506,-176.079,7.409,148.262
C02355=1218.361,342.181,-72.538,-176.077,7.412,148.262
C02356=1218.356,342.429,-72.570,-176.075,7.414,148.262
C02357=1218.352,342.677,-72.601,-176.073,7.418,148.262
C02358=1218.348,342.926,-72.633,-176.071,7.420,148.263
C02359=1218.343,343.173,-72.665,-176.070,7.423,148.263
C02360=1218.340,343.421,-72.697,-176.067,7.426,148.263
C02361=1218.335,343.669,-72.729,-176.066,7.429,148.263
C02362=1218.331,343.917,-72.761,-176.063,7.432,148.263
C02363=1218.327,344.165,-72.792,-176.061,7.434,148.263
C02364=1218.322,344.412,-72.825,-176.059,7.438,148.264
C02365=1218.318,344.660,-72.856,-176.058,7.440,148.264
C02366=1218.314,344.909,-72.889,-176.056,7.443,148.264
C02367=1218.311,345.156,-72.921,-176.054,7.446,148.264
C02368=1218.306,345.403,-72.953,-176.052,7.449,148.264
C02369=1218.302,345.652,-72.985,-176.050,7.452,148.265
C02370=1218.298,345.900,-73.017,-176.048,7.454,148.265
C02371=1218.293,346.147,-73.049,-176.047,7.457,148.265
C02372=1218.289,346.395,-73.081,-176.044,7.460,148.265
C02373=1218.285,346.644,-73.113,-176.042,7.463,148.265
C02374=1218.281,346.891,-73.145,-176.040,7.466,148.265
C02375=1218.276,347.140,-73.177,-176.039,7.468,148.266
C02376=1218.273,347.387,-73.210,-176.037,7.471,148.266
C02377=1218.268,347.635,-73.242,-176.035,7.474,148.266
C02378=1218.264,347.883,-73.274,-176.033,7.477,148.266
C02379=1218.260,348.131,-73.306,-176.031,7.480,148.266
C02380=1218.256,348.379,-73.338,-176.029,7.483,148.267
C02381=1218.251,348.627,-73.370,-176.028,7.485,148.267
C02382=1218.247,348.874,-73.403,-176.025,7.489,148.267
C02383=1218.243,349.122,-73.435,-176.024,7.491,148.267
C02384=1218.239,349.370,-73.467,-176.022,7.494,148.267
C02385=1218.234,349.618,-73.499,-176.020,7.497,148.268
C02386=1218.231,349.866,-73.532,-176.018,7.500,148.268
C02387=1218.226,350.114,-73.564,-176.017,7.503,148.268
C02388=1218.223,350.362,-73.596,-176.015,7.506,148.268
C02389=1218.219,350.610,-73.629,-176.013,7.508,148.269
C02390=1218.214,350.857,-73.661,-176.011,7.512,148.269
C02391=1218.210,351.105,-73.693,-176.009,7.514,148.269
C02392=1218.206,351.353,-73.726,-176.007,7.517,148.269
C02393=1218.202,351.601,-73.758,-176.006,7.520,148.269
C02394=1218.197,351.849,-73.790,-176.004,7.522,148.270
C02395=1218.193,352.096,-73.823,-176.002,7.526,148.270
C02396=1218.189,352.345,-73.855,-176.000,7.528,148.270
C02397=1218.185,352.593,-73.888,-175.999,7.531,148.270
C02398=1218.181,352.840,-73.920,-175.997,7.535,148.271
C02399=1218.177,353.089,-73.953,-175.995,7.537,148.271
C02400=1218.173,353.335,-73.985,-175.993,7.540,148.271
C02401=1218.168,353.584,-74.017,-175.991,7.543,148.271
C02402=1218.164,353.832,-74.050,-175.990,7.545,148.271
C02403=1218.160,354.079,-74.082,-175.988,7.549,148.272
C02404=1218.156,354.328,-74.115,-175.986,7.552,148.272
C02405=1218.151,354.575,-74.147,-175.985,7.554,148.272
C02406=1218.148,354.823,-74.179,-175.982,7.558,148.272
C02407=1218.143,355.071,-74.212,-175.981,7.560,148.273
C02408=1218.139,355.319,-74.245,-175.980,7.563,148.273
C02409=1218.135,355.567,-74.278,-175.977,7.566,148.273
C02410=1218.131,355.815,-74.310,-175.976,7.569,148.273
C02411=1218.127,356.062,-74.343,-175.974,7.571,148.274
C02412=1218.122,356.310,-74.375,-175.972,7.575,148.274
C02413=1218.119,356.558,-74.408,-175.971,7.577,148.274
C02414=1218.114,356.806,-74.440,-175.969,7.580,148.274
C02415=1218.110,357.054,-74.473,-175.967,7.583,148.275
C02416=1218.106,357.301,-74.506,-175.966,7.586,148.275
C02417=1218.102,357.549,-74.538,-175.964,7.589,148.275
C02418=1218.098,357.797,-74.571,-175.962,7.592,148.275
C02419=1218.094,358.045,-74.604,-175.961,7.595,148.276
C02420=1218.089,358.293,-74.637,-175.959,7.597,148.276
C02421=1218.085,358.540,-74.669,-175.957,7.601,148.276
C02422=1218.081,358.788,-74.702,-175.956,7.604,148.277
C02423=1218.077,359.036,-74.735,-175.954,7.606,148.277
C02424=1218.073,359.284,-74.768,-175.952,7.609,148.277
C02425=1218.069,359.532,-74.800,-175.951,7.612,148.277
C02426=1218.065,359.779,-74.833,-175.949,7.615,148.278
C02427=1218.061,360.027,-74.866,-175.948,7.618,148.278
C02428=1218.056,360.276,-74.899,-175.946,7.621,148.278
C02429=1218.052,360.523,-74.932,-175.944,7.623,148.278
C02430=1218.048,360.771,-74.965,-175.943,7.626,148.279
C02431=1218.045,361.018,-74.997,-175.941,7.630,148.279
C02432=1218.040,361.267,-75.030,-175.939,7.632,148.279
C02433=1218.036,361.515,-75.063,-175.938,7.635,148.280
C02434=1218.032,361.762,-75.096,-175.937,7.638,148.280
C02435=1218.028,362.010,-75.129,-175.934,7.641,148.280
C02436=1218.024,362.258,-75.163,-175.933,7.644,148.280
C02437=1218.019,362.505,-75.195,-175.932,7.646,148.281
C02438=1218.015,362.753,-75.227,-175.929,7.650,148.281
C02439=1218.011,363.001,-75.260,-175.928,7.653,148.281
C02440=1218.007,363.248,-75.293,-175.927,7.655,148.282
C02441=1218.003,363.496,-75.327,-175.925,7.658,148.282
C02442=1217.999,363.744,-75.360,-175.923,7.661,148.282
C02443=1217.994,363.992,-75.392,-175.922,7.664,148.283
C02444=1217.990,364.240,-75.425,-175.921,7.667,148.283
C02445=1217.986,364.488,-75.459,-175.919,7.670,148.283
C02446=1217.982,364.735,-75.492,-175.918,7.672,148.284
C02447=1217.978,364.983,-75.525,-175.916,7.676,148.284
C02448=1217.973,365.231,-75.558,-175.915,7.679,148.284
C02449=1217.970,365.478,-75.591,-175.913,7.681,148.284
C02450=1217.966,365.726,-75.624,-175.912,7.684,148.285
C02451=1217.962,365.974,-75.657,-175.910,7.687,148.285
C02452=1217.958,366.221,-75.690,-175.908,7.690,148.286
C02453=1217.954,366.470,-75.724,-175.907,7.693,148.286
C02454=1217.949,366.750,-75.760,-175.906,7.696,148.286
C02455=1217.944,367.030,-75.798,-175.904,7.699,148.287
C02456=1217.939,367.309,-75.836,-175.902,7.703,148.287
C02457=1217.934,367.590,-75.873,-175.901,7.705,148.287
C02458=1217.930,367.837,-75.906,-175.899,7.709,148.288
C02459=1217.927,368.086,-75.940,-175.898,7.712,148.288
C02460=1217.923,368.334,-75.973,-175.896,7.714,148.288
C02461=1217.918,368.581,-76.006,-175.895,7.717,148.289
C02462=1217.915,368.828,-76.040,-175.894,7.720,148.289
C02463=1217.910,369.076,-76.073,-175.892,7.723,148.289
C02464=1217.906,369.324,-76.106,-175.891,7.725,148.290
C02465=1217.902,369.572,-76.139,-175.889,7.729,148.290
C02466=1217.898,369.819,-76.172,-175.888,7.732,148.290
C02467=1217.894,370.067,-76.205,-175.887,7.734,148.291
C02468=1217.890,370.315,-76.239,-175.885,7.737,148.291
C02469=1217.886,370.562,-76.272,-175.884,7.740,148.292
C02470=1217.881,370.810,-76.305,-175.883,7.743,148.292
C02471=1217.877,371.058,-76.338,-175.881,7.745,148.292
C02472=1217.873,371.305,-76.373,-175.880,7.748,148.293
C02473=1217.869,371.554,-76.406,-175.879,7.751,148.293
C02474=1217.865,371.802,-76.439,-175.877,7.755,148.293
C02475=1217.861,372.049,-76.472,-175.876,7.758,148.294
C02476=1217.857,372.297,-76.506,-175.875,7.760,148.294
C02477=1217.853,372.545,-76.539,-175.873,7.763,148.294
C02478=1217.849,372.792,-76.573,-175.872,7.766,148.295
C02479=1217.845,373.040,-76.606,-175.871,7.769,148.295
C02480=1217.840,373.288,-76.639,-175.870,7.771,148.296
C02481=1217.836,373.535,-76.673,-175.869,7.774,148.296
C02482=1217.832,373.784,-76.706,-175.867,7.777,148.296
C02483=1217.828,374.031,-76.740,-175.866,7.780,148.297
C02484=1217.824,374.279,-76.773,-175.865,7.783,148.297
C02485=1217.820,374.526,-76.806,-175.864,7.785,148.298
C02486=1217.815,374.774,-76.841,-175.863,7.788,148.298
C02487=1217.811,375.021,-76.874,-175.861,7.791,148.298
C02488=1217.807,375.269,-76.907,-175.860,7.794,148.299
C02489=1217.803,375.517,-76.940,-175.859,7.796,148.299
C02490=1217.800,375.765,-76.975,-175.857,7.799,148.299
C02491=1217.796,376.012,-77.008,-175.856,7.802,148.300
C02492=1217.791,376.260,-77.041,-175.855,7.805,148.300
C02493=1217.787,376.508,-77.075,-175.854,7.808,148.300
C02494=1217.783,376.755,-77.108,-175.853,7.810,148.301
C02495=1217.779,377.003,-77.142,-175.852,7.813,148.301
C02496=1217.775,377.251,-77.176,-175.850,7.816,148.302
C02497=1217.771,377.499,-77.210,-175.850,7.819,148.302
C02498=1217.766,377.747,-77.243,-175.848,7.822,148.303
C02499=1217.763,377.994,-77.277,-175.847,7.825,148.303
C02500=1217.758,378.242,-77.310,-175.846,7.828,148.303
C02501=1217.755,378.490,-77.345,-175.845,7.830,148.304
C02502=1217.750,378.737,-77.378,-175.844,7.833,148.304
C02503=1217.747,378.984,-77.412,-175.842,7.836,148.305
C02504=1217.742,379.232,-77.445,-175.842,7.838,148.305
C02505=1217.738,379.480,-77.479,-175.841,7.841,148.305
C02506=1217.734,379.727,-77.512,-175.839,7.844,148.306
C02507=1217.729,379.976,-77.547,-175.838,7.847,148.306
C02508=1217.726,380.223,-77.580,-175.837,7.849,148.307
C02509=1217.721,380.471,-77.614,-175.836,7.852,148.307
C02510=1217.718,380.718,-77.647,-175.835,7.855,148.308
C02511=1217.713,380.967,-77.682,-175.834,7.858,148.308
C02512=1217.710,381.214,-77.715,-175.833,7.860,148.308
C02513=1217.705,381.462,-77.749,-175.832,7.863,148.309
C02514=1217.701,381.709,-77.783,-175.831,7.866,148.309
C02515=1217.697,381.957,-77.816,-175.830,7.869,148.310
C02516=1217.693,382.205,-77.850,-175.829,7.872,148.310
C02517=1217.689,382.453,-77.884,-175.828,7.874,148.310
C02518=1217.685,382.700,-77.918,-175.827,7.876,148.311
C02519=1217.681,382.947,-77.951,-175.826,7.879,148.311
C02520=1217.677,383.196,-77.986,-175.825,7.882,148.312
C02521=1217.673,383.443,-78.019,-175.824,7.885,148.312
C02522=1217.668,383.691,-78.054,-175.823,7.888,148.313
C02523=1217.664,383.938,-78.088,-175.822,7.890,148.313
C02524=1217.661,384.186,-78.121,-175.821,7.893,148.313
C02525=1217.656,384.434,-78.156,-175.820,7.896,148.314
C02526=1217.652,384.681,-78.189,-175.819,7.899,148.314
C02527=1217.648,384.928,-78.223,-175.818,7.902,148.315
C02528=1217.644,385.177,-78.257,-175.817,7.904,148.315
C02529=1217.640,385.424,-78.291,-175.817,7.907,148.316
C02530=1217.635,385.672,-78.325,-175.815,7.909,148.316
C02531=1217.632,385.919,-78.359,-175.815,7.911,148.316
C02532=1217.627,386.168,-78.393,-175.814,7.914,148.317
C02533=1217.623,386.415,-78.427,-175.813,7.917,148.317
C02534=1217.620,386.662,-78.461,-175.812,7.920,148.318
C02535=1217.615,386.911,-78.495,-175.811,7.922,148.318
C02536=1217.611,387.158,-78.529,-175.810,7.925,148.319
C02537=1217.607,387.405,-78.563,-175.809,7.928,148.319
C02538=1217.603,387.653,-78.596,-175.808,7.930,148.319
C02539=1217.599,387.901,-78.631,-175.808,7.933,148.320
C02540=1217.595,388.148,-78.665,-175.807,7.936,148.320
C02541=1217.590,388.396,-78.699,-175.806,7.938,148.321
C02542=1217.587,388.644,-78.733,-175.805,7.941,148.321
C02543=1217.583,388.891,-78.767,-175.804,7.944,148.322
C02544=1217.578,389.138,-78.801,-175.803,7.946,148.322
C02545=1217.575,389.387,-78.835,-175.803,7.949,148.323
C02546=1217.570,389.634,-78.869,-175.801,7.952,148.323
C02547=1217.567,389.881,-78.903,-175.801,7.954,148.323
C02548=1217.563,390.130,-78.938,-175.800,7.957,148.324
C02549=1217.559,390.377,-78.972,-175.799,7.960,148.324
C02550=1217.554,390.625,-79.006,-175.798,7.962,148.325
C02551=1217.551,390.872,-79.040,-175.797,7.965,148.325
C02552=1217.546,391.120,-79.074,-175.797,7.967,148.326
C02553=1217.542,391.367,-79.108,-175.796,7.970,148.326
C02554=1217.538,391.615,-79.143,-175.795,7.973,148.327
C02555=1217.534,391.863,-79.176,-175.794,7.975,148.327
C02556=1217.530,392.110,-79.211,-175.793,7.978,148.328
C02557=1217.526,392.358,-79.245,-175.793,7.980,148.328
C02558=1217.521,392.640,-79.284,-175.792,7.983,148.329
C02559=1217.516,392.922,-79.323,-175.791,7.986,148.329
C02560=1217.512,393.203,-79.362,-175.790,7.989,148.330
C02561=1217.507,393.486,-79.401,-175.789,7.992,148.330
C02562=1217.504,393.733,-79.435,-175.789,7.994,148.331
C02563=1217.499,393.981,-79.469,-175.788,7.997,148.331
C02564=1217.495,394.229,-79.504,-175.787,7.999,148.331
C02565=1217.491,394.476,-79.538,-175.786,8.002,148.332
C02566=1217.487,394.723,-79.573,-175.786,8.004,148.332
C02567=1217.484,394.971,-79.607,-175.785,8.007,148.333
C02568=1217.479,395.219,-79.641,-175.785,8.009,148.333
C02569=1217.475,395.466,-79.674,-175.783,8.012,148.334
C02570=1217.471,395.715,-79.709,-175.783,8.014,148.334
C02571=1217.466,395.962,-79.744,-175.782,8.017,148.335
C02572=1217.463,396.210,-79.778,-175.782,8.019,148.335
C02573=1217.458,396.457,-79.812,-175.781,8.022,148.336
C02574=1217.454,396.705,-79.847,-175.780,8.024,148.336
C02575=1217.451,396.952,-79.881,-175.779,8.027,148.337
C02576=1217.446,397.200,-79.916,-175.779,8.029,148.337
C02577=1217.442,397.447,-79.950,-175.778,8.031,148.337
C02578=1217.438,397.695,-79.984,-175.777,8.034,148.338
C02579=1217.434,397.942,-80.019,-175.777,8.037,148.338
C02580=1217.430,398.190,-80.053,-175.776,8.039,148.339
C02581=1217.426,398.438,-80.088,-175.776,8.042,148.339
C02582=1217.422,398.686,-80.122,-175.775,8.044,148.340
C02583=1217.418,398.933,-80.156,-175.774,8.047,148.340
C02584=1217.414,399.180,-80.191,-175.774,8.049,148.341
C02585=1217.410,399.428,-80.226,-175.773,8.052,148.341
C02586=1217.406,399.676,-80.259,-175.772,8.054,148.342
C02587=1217.402,399.924,-80.294,-175.772,8.056,148.342
C02588=1217.397,400.171,-80.329,-175.771,8.059,148.342
C02589=1217.393,400.418,-80.363,-175.771,8.061,148.343
C02590=1217.389,400.666,-80.397,-175.770,8.063,148.343
C02591=1217.385,400.913,-80.433,-175.769,8.066,148.344
C02592=1217.382,401.161,-80.467,-175.769,8.068,148.344
C02593=1217.377,401.408,-80.501,-175.768,8.070,148.345
C02594=1217.373,401.656,-80.536,-175.767,8.073,148.345
C02595=1217.370,401.904,-80.570,-175.767,8.076,148.346
C02596=1217.365,402.151,-80.604,-175.766,8.078,148.346
C02597=1217.361,402.399,-80.639,-175.766,8.081,148.347
C02598=1217.357,402.646,-80.673,-175.765,8.083,148.347
C02599=1217.353,402.894,-80.708,-175.765,8.085,148.348
C02600=1217.349,403.142,-80.742,-175.764,8.087,148.348
C02601=1217.345,403.389,-80.778,-175.763,8.090,148.348
C02602=1217.341,403.636,-80.812,-175.763,8.092,148.349
C02603=1217.337,403.885,-80.847,-175.763,8.094,148.349
C02604=1217.333,404.132,-80.881,-175.761,8.097,148.350
C02605=1217.329,404.380,-80.915,-175.761,8.099,148.350
C02606=1217.325,404.627,-80.950,-175.761,8.101,148.351
C02607=1217.321,404.874,-80.985,-175.760,8.104,148.351
C02608=1217.317,405.122,-81.020,-175.759,8.106,148.352
C02609=1217.313,405.369,-81.054,-175.759,8.109,148.352
C02610=1217.309,405.617,-81.089,-175.758,8.111,148.352
C02611=1217.304,405.865,-81.123,-175.758,8.113,148.353
C02612=1217.300,406.113,-81.158,-175.757,8.115,148.353
C02613=1217.297,406.359,-81.192,-175.757,8.118,148.354
C02614=1217.293,406.607,-81.227,-175.756,8.120,148.354
C02615=1217.288,406.855,-81.262,-175.756,8.122,148.355
C02616=1217.284,407.103,-81.297,-175.755,8.124,148.355
C02617=1217.280,407.350,-81.332,-175.755,8.126,148.356
C02618=1217.277,407.598,-81.366,-175.754,8.129,148.356
C02619=1217.272,407.845,-81.401,-175.754,8.132,148.357
C02620=1217.268,408.093,-81.435,-175.753,8.133,148.357
C02621=1217.264,408.340,-81.471,-175.753,8.136,148.357
C02622=1217.260,408.588,-81.505,-175.752,8.138,148.358
C02623=1217.256,408.835,-81.539,-175.751,8.141,148.358
C02624=1217.252,409.083,-81.574,-175.751,8.143,148.359
C02625=1217.248,409.330,-81.609,-175.751,8.145,148.359
C02626=1217.244,409.578,-81.644,-175.750,8.147,148.360
C02627=1217.239,409.826,-81.679,-175.750,8.149,148.360
C02628=1217.236,410.073,-81.713,-175.749,8.151,148.360
C02629=1217.232,410.320,-81.748,-175.749,8.154,148.361
C02630=1217.228,410.568,-81.783,-175.748,8.156,148.361
C02631=1217.223,410.816,-81.817,-175.747,8.159,148.362
C02632=1217.220,411.063,-81.853,-175.747,8.161,148.362
C02633=1217.216,411.310,-81.887,-175.747,8.163,148.363
C02634=1217.212,411.559,-81.922,-175.746,8.165,148.363
C02635=1217.208,411.806,-81.957,-175.746,8.167,148.364
C02636=1217.204,412.053,-81.992,-175.745,8.169,148.364
C02637=1217.200,412.302,-82.026,-175.745,8.171,148.365
C02638=1217.195,412.548,-82.062,-175.744,8.173,148.365
C02639=1217.191,412.796,-82.096,-175.744,8.176,148.365
C02640=1217.188,413.044,-82.130,-175.743,8.178,148.366
C02641=1217.184,413.291,-82.166,-175.743,8.181,148.366
C02642=1217.179,413.539,-82.200,-175.742,8.183,148.367
C02643=1217.176,413.786,-82.236,-175.742,8.185,148.367
C02644=1217.171,414.033,-82.270,-175.741,8.187,148.368
C02645=1217.167,414.282,-82.305,-175.741,8.189,148.368
C02646=1217.163,414.528,-82.340,-175.740,8.191,148.368
C02647=1217.159,414.776,-82.375,-175.740,8.193,148.369
C02648=1217.156,415.024,-82.410,-175.739,8.195,148.369
C02649=1217.151,415.271,-82.445,-175.739,8.198,148.370
C02650=1217.147,415.498,-82.477,-175.739,8.200,148.370
C02651=1217.144,415.726,-82.508,-175.738,8.202,148.371
C02652=1217.140,415.953,-82.541,-175.738,8.204,148.371
C02653=1217.136,416.181,-82.573,-175.737,8.206,148.371
C02654=1217.133,416.408,-82.605,-175.737,8.207,148.372
C02655=1217.129,416.635,-82.637,-175.737,8.209,148.372
C02656=1217.127,416.864,-82.669,-175.736,8.211,148.373
C02657=1217.127,417.090,-82.701,-175.735,8.213,148.373
C02658=1216.706,417.090,-82.736,-175.739,8.224,148.377
C02659=1216.705,416.862,-82.704,-175.740,8.222,148.376
C02660=1216.706,416.633,-82.672,-175.740,8.220,148.376
C02661=1216.710,416.404,-82.640,-175.740,8.218,148.375
C02662=1216.715,416.175,-82.608,-175.740,8.217,148.375
C02663=1216.718,415.947,-82.575,-175.741,8.215,148.375
C02664=1216.722,415.718,-82.543,-175.741,8.212,148.374
C02665=1216.725,415.489,-82.510,-175.742,8.210,148.374
C02666=1216.729,415.261,-82.478,-175.742,8.208,148.373
C02667=1216.733,415.014,-82.443,-175.743,8.206,148.373
C02668=1216.737,414.766,-82.408,-175.743,8.204,148.373
C02669=1216.741,414.518,-82.374,-175.744,8.202,148.372
C02670=1216.746,414.271,-82.338,-175.744,8.200,148.372
C02671=1216.750,414.023,-82.304,-175.745,8.198,148.371
C02672=1216.754,413.776,-82.268,-175.745,8.196,148.371
C02673=1216.757,413.528,-82.234,-175.745,8.193,148.370
C02674=1216.762,413.281,-82.200,-175.746,8.191,148.370
C02675=1216.765,413.033,-82.164,-175.746,8.189,148.370
C02676=1216.770,412.786,-82.130,-175.747,8.186,148.369
C02677=1216.774,412.538,-82.095,-175.748,8.184,148.369
C02678=1216.778,412.291,-82.060,-175.748,8.182,148.368
C02679=1216.782,412.043,-82.025,-175.749,8.180,148.368
C02680=1216.785,411.795,-81.991,-175.749,8.178,148.367
C02681=1216.790,411.548,-81.955,-175.749,8.176,148.367
C02682=1216.794,411.300,-81.921,-175.750,8.173,148.366
C02683=1216.798,411.052,-81.886,-175.750,8.171,148.366
C02684=1216.802,410.805,-81.851,-175.750,8.169,148.366
C02685=1216.806,410.558,-81.816,-175.751,8.167,148.365
C02686=1216.810,410.310,-81.782,-175.752,8.164,148.365
C02687=1216.814,410.063,-81.747,-175.752,8.162,148.364
C02688=1216.818,409.815,-81.712,-175.753,8.160,148.364
C02689=1216.822,409.567,-81.677,-175.753,8.158,148.363
C02690=1216.826,409.320,-81.642,-175.753,8.155,148.363
C02691=1216.831,409.072,-81.607,-175.754,8.153,148.363
C02692=1216.834,408.825,-81.573,-175.754,8.151,148.362
C02693=1216.838,408.577,-81.539,-175.756,8.148,148.362
C02694=1216.842,408.330,-81.503,-175.756,8.146,148.361
C02695=1216.847,408.082,-81.469,-175.756,8.144,148.361
C02696=1216.851,407.834,-81.434,-175.757,8.142,148.360
C02697=1216.854,407.588,-81.399,-175.757,8.140,148.360
C02698=1216.858,407.340,-81.364,-175.757,8.138,148.359
C02699=1216.863,407.092,-81.330,-175.759,8.135,148.359
C02700=1216.867,406.844,-81.295,-175.759,8.133,148.358
C02701=1216.871,406.597,-81.261,-175.759,8.131,148.358
C02702=1216.874,406.349,-81.226,-175.760,8.128,148.357
C02703=1216.879,406.102,-81.191,-175.760,8.126,148.357
C02704=1216.883,405.854,-81.156,-175.761,8.123,148.357
C02705=1216.887,405.606,-81.122,-175.762,8.121,148.356
C02706=1216.890,405.359,-81.087,-175.762,8.119,148.356
C02707=1216.895,405.112,-81.053,-175.763,8.117,148.355
C02708=1216.899,404.864,-81.018,-175.763,8.114,148.355
C02709=1216.903,404.616,-80.983,-175.764,8.112,148.354
C02710=1216.907,404.369,-80.949,-175.764,8.110,148.354
C02711=1216.911,404.121,-80.915,-175.764,8.107,148.353
C02712=1216.915,403.874,-80.879,-175.766,8.105,148.353
C02713=1216.919,403.626,-80.845,-175.766,8.102,148.352
C02714=1216.923,403.379,-80.811,-175.766,8.100,148.352
C02715=1216.927,403.131,-80.776,-175.767,8.098,148.351
C02716=1216.932,402.884,-80.741,-175.768,8.095,148.351
C02717=1216.935,402.636,-80.707,-175.768,8.093,148.351
C02718=1216.940,402.388,-80.673,-175.769,8.091,148.350
C02719=1216.943,402.141,-80.637,-175.769,8.088,148.350
C02720=1216.948,401.893,-80.603,-175.770,8.086,148.349
C02721=1216.951,401.646,-80.568,-175.770,8.084,148.349
C02722=1216.956,401.398,-80.534,-175.771,8.081,148.348
C02723=1216.960,401.151,-80.499,-175.772,8.079,148.348
C02724=1216.963,400.903,-80.465,-175.772,8.077,148.347
C02725=1216.968,400.656,-80.431,-175.773,8.073,148.347
C02726=1216.972,400.407,-80.396,-175.774,8.071,148.347
C02727=1216.976,400.160,-80.362,-175.774,8.069,148.346
C02728=1216.980,399.912,-80.327,-175.775,8.066,148.346
C02729=1216.984,399.665,-80.293,-175.775,8.064,148.345
C02730=1216.988,399.418,-80.259,-175.776,8.062,148.345
C02731=1216.992,399.170,-80.224,-175.777,8.059,148.344
C02732=1216.996,398.923,-80.189,-175.777,8.057,148.344
C02733=1217.000,398.675,-80.155,-175.777,8.055,148.343
C02734=1217.004,398.427,-80.120,-175.779,8.052,148.343
C02735=1217.008,398.179,-80.085,-175.779,8.050,148.342
C02736=1217.012,397.932,-80.051,-175.780,8.047,148.342
C02737=1217.016,397.685,-80.017,-175.780,8.045,148.341
C02738=1217.020,397.437,-79.982,-175.781,8.042,148.341
C02739=1217.024,397.190,-79.948,-175.782,8.040,148.340
C02740=1217.028,396.941,-79.913,-175.782,8.038,148.340
C02741=1217.032,396.694,-79.880,-175.783,8.034,148.340
C02742=1217.037,396.447,-79.845,-175.784,8.032,148.339
C02743=1217.041,396.198,-79.811,-175.784,8.029,148.339
C02744=1217.045,395.951,-79.777,-175.785,8.027,148.338
C02745=1217.049,395.704,-79.743,-175.786,8.025,148.338
C02746=1217.053,395.456,-79.708,-175.786,8.022,148.337
C02747=1217.057,395.208,-79.674,-175.788,8.019,148.337
C02748=1217.061,394.960,-79.639,-175.788,8.017,148.336
C02749=1217.065,394.713,-79.605,-175.789,8.014,148.336
C02750=1217.070,394.466,-79.571,-175.789,8.012,148.335
C02751=1217.073,394.218,-79.537,-175.790,8.009,148.335
C02752=1217.077,393.971,-79.502,-175.791,8.007,148.334
C02753=1217.081,393.722,-79.467,-175.792,8.004,148.334
C02754=1217.085,393.475,-79.433,-175.792,8.002,148.334
C02755=1217.090,393.193,-79.395,-175.793,7.999,148.333
C02756=1217.094,392.912,-79.356,-175.794,7.996,148.333
C02757=1217.099,392.629,-79.317,-175.795,7.993,148.332
C02758=1217.104,392.347,-79.277,-175.796,7.990,148.332
C02759=1217.108,392.100,-79.243,-175.796,7.988,148.331
C02760=1217.112,391.853,-79.209,-175.797,7.985,148.331
C02761=1217.116,391.604,-79.175,-175.798,7.983,148.330
C02762=1217.120,391.357,-79.141,-175.799,7.980,148.330
C02763=1217.124,391.110,-79.107,-175.800,7.977,148.329
C02764=1217.128,390.862,-79.072,-175.800,7.975,148.329
C02765=1217.132,390.614,-79.038,-175.801,7.972,148.328
C02766=1217.136,390.366,-79.004,-175.802,7.970,148.328
C02767=1217.140,390.119,-78.970,-175.803,7.967,148.327
C02768=1217.145,389.871,-78.936,-175.804,7.964,148.327
C02769=1217.149,389.624,-78.902,-175.804,7.962,148.327
C02770=1217.153,389.376,-78.867,-175.805,7.959,148.326
C02771=1217.157,389.128,-78.834,-175.806,7.957,148.326
C02772=1217.161,388.881,-78.800,-175.807,7.954,148.325
C02773=1217.164,388.633,-78.765,-175.808,7.951,148.325
C02774=1217.169,388.386,-78.731,-175.808,7.949,148.324
C02775=1217.173,388.138,-78.698,-175.810,7.946,148.324
C02776=1217.177,387.890,-78.663,-175.810,7.943,148.323
C02777=1217.181,387.643,-78.629,-175.811,7.941,148.323
C02778=1217.186,387.395,-78.595,-175.812,7.938,148.323
C02779=1217.189,387.147,-78.561,-175.813,7.935,148.322
C02780=1217.193,386.900,-78.527,-175.814,7.932,148.322
C02781=1217.197,386.652,-78.493,-175.815,7.931,148.321
C02782=1217.202,386.404,-78.460,-175.815,7.927,148.321
C02783=1217.206,386.156,-78.425,-175.817,7.925,148.320
C02784=1217.209,385.909,-78.391,-175.817,7.923,148.320
C02785=1217.214,385.661,-78.357,-175.818,7.920,148.319
C02786=1217.218,385.413,-78.323,-175.819,7.917,148.319
C02787=1217.221,385.166,-78.289,-175.820,7.914,148.319
C02788=1217.226,384.918,-78.255,-175.821,7.912,148.318
C02789=1217.230,384.671,-78.221,-175.822,7.909,148.318
C02790=1217.234,384.422,-78.187,-175.823,7.906,148.317
C02791=1217.238,384.175,-78.153,-175.824,7.903,148.317
C02792=1217.242,383.928,-78.119,-175.825,7.900,148.316
C02793=1217.247,383.680,-78.086,-175.825,7.898,148.316
C02794=1217.250,383.432,-78.051,-175.827,7.895,148.316
C02795=1217.255,383.184,-78.018,-175.828,7.892,148.315
C02796=1217.259,382.937,-77.984,-175.829,7.890,148.315
C02797=1217.263,382.690,-77.950,-175.830,7.886,148.314
C02798=1217.267,382.441,-77.916,-175.830,7.885,148.314
C02799=1217.271,382.194,-77.882,-175.832,7.882,148.313
C02800=1217.275,381.947,-77.849,-175.833,7.879,148.313
C02801=1217.279,381.699,-77.814,-175.834,7.876,148.313
C02802=1217.283,381.451,-77.781,-175.835,7.873,148.312
C02803=1217.287,381.204,-77.747,-175.836,7.870,148.312
C02804=1217.292,380.956,-77.713,-175.837,7.868,148.311
C02805=1217.296,380.708,-77.679,-175.838,7.865,148.311
C02806=1217.300,380.461,-77.646,-175.839,7.863,148.311
C02807=1217.304,380.213,-77.611,-175.840,7.860,148.310
C02808=1217.308,379.965,-77.578,-175.841,7.857,148.310
C02809=1217.312,379.718,-77.544,-175.843,7.854,148.309
C02810=1217.316,379.470,-77.511,-175.843,7.851,148.309
C02811=1217.320,379.222,-77.476,-175.844,7.848,148.308
C02812=1217.324,378.974,-77.443,-175.846,7.845,148.308
C02813=1217.328,378.726,-77.410,-175.846,7.843,148.308
C02814=1217.333,378.479,-77.376,-175.847,7.841,148.307
C02815=1217.337,378.231,-77.342,-175.849,7.838,148.307
C02816=1217.341,377.984,-77.309,-175.850,7.835,148.306
C02817=1217.344,377.736,-77.275,-175.851,7.832,148.306
C02818=1217.349,377.488,-77.241,-175.852,7.829,148.306
C02819=1217.353,377.241,-77.207,-175.853,7.826,148.305
C02820=1217.357,376.993,-77.174,-175.855,7.824,148.305
C02821=1217.361,376.746,-77.140,-175.856,7.821,148.304
C02822=1217.365,376.497,-77.106,-175.857,7.818,148.304
C02823=1217.369,376.249,-77.073,-175.858,7.815,148.304
C02824=1217.373,376.002,-77.039,-175.859,7.812,148.303
C02825=1217.377,375.754,-77.006,-175.861,7.810,148.303
C02826=1217.381,375.507,-76.973,-175.862,7.807,148.302
C02827=1217.386,375.259,-76.938,-175.863,7.804,148.302
C02828=1217.390,375.012,-76.905,-175.864,7.801,148.302
C02829=1217.394,374.763,-76.872,-175.865,7.798,148.301
C02830=1217.398,374.515,-76.839,-175.866,7.795,148.301
C02831=1217.401,374.268,-76.805,-175.868,7.793,148.301
C02832=1217.406,374.020,-76.771,-175.869,7.790,148.300
C02833=1217.411,373.773,-76.738,-175.870,7.787,148.300
C02834=1217.415,373.525,-76.705,-175.871,7.784,148.299
C02835=1217.418,373.278,-76.671,-175.872,7.781,148.299
C02836=1217.422,373.029,-76.637,-175.874,7.779,148.299
C02837=1217.426,372.782,-76.604,-175.875,7.776,148.298
C02838=1217.430,372.534,-76.571,-175.876,7.773,148.298
C02839=1217.435,372.286,-76.537,-175.878,7.770,148.298
C02840=1217.439,372.039,-76.503,-175.879,7.768,148.297
C02841=1217.443,371.791,-76.470,-175.881,7.764,148.297
C02842=1217.447,371.543,-76.437,-175.882,7.761,148.296
C02843=1217.451,371.295,-76.404,-175.883,7.758,148.296
C02844=1217.456,371.048,-76.371,-175.884,7.755,148.296
C02845=1217.459,370.800,-76.337,-175.886,7.753,148.295
C02846=1217.463,370.552,-76.303,-175.887,7.750,148.295
C02847=1217.467,370.304,-76.270,-175.888,7.747,148.295
C02848=1217.472,370.056,-76.236,-175.889,7.745,148.294
C02849=1217.476,369.809,-76.203,-175.890,7.742,148.294
C02850=1217.480,369.561,-76.170,-175.893,7.738,148.294
C02851=1217.484,369.313,-76.137,-175.894,7.736,148.293
C02852=1217.488,369.065,-76.104,-175.895,7.733,148.293
C02853=1217.493,368.818,-76.071,-175.896,7.730,148.292
C02854=1217.497,368.570,-76.038,-175.898,7.727,148.292
C02855=1217.501,368.323,-76.004,-175.899,7.725,148.292
C02856=1217.505,368.075,-75.970,-175.901,7.721,148.291
C02857=1217.509,367.827,-75.937,-175.902,7.718,148.291
C02858=1217.513,367.580,-75.904,-175.904,7.716,148.291
C02859=1217.517,367.299,-75.867,-175.905,7.713,148.290
C02860=1217.522,367.019,-75.829,-175.907,7.709,148.290
C02861=1217.527,366.740,-75.792,-175.909,7.706,148.290
C02862=1217.532,366.459,-75.755,-175.910,7.703,148.289
C02863=1217.536,366.211,-75.721,-175.912,7.699,148.289
C02864=1217.540,365.964,-75.689,-175.913,7.697,148.289
C02865=1217.544,365.716,-75.656,-175.914,7.694,148.288
C02866=1217.548,365.469,-75.623,-175.916,7.691,148.288
C02867=1217.552,365.221,-75.589,-175.917,7.689,148.288
C02868=1217.556,364.972,-75.556,-175.919,7.685,148.287
C02869=1217.560,364.725,-75.523,-175.921,7.682,148.287
C02870=1217.564,364.477,-75.490,-175.922,7.680,148.287
C02871=1217.568,364.229,-75.456,-175.923,7.677,148.286
C02872=1217.572,363.981,-75.423,-175.925,7.673,148.286
C02873=1217.576,363.734,-75.390,-175.926,7.671,148.286
C02874=1217.581,363.485,-75.358,-175.928,7.668,148.285
C02875=1217.585,363.238,-75.324,-175.929,7.665,148.285
C02876=1217.590,362.991,-75.292,-175.931,7.662,148.285
C02877=1217.594,362.743,-75.259,-175.933,7.659,148.284
C02878=1217.597,362.495,-75.226,-175.934,7.657,148.284
C02879=1217.601,362.248,-75.193,-175.935,7.654,148.284
C02880=1217.606,361.999,-75.160,-175.938,7.650,148.284
C02881=1217.610,361.752,-75.127,-175.939,7.648,148.283
C02882=1217.614,361.504,-75.094,-175.940,7.645,148.283
C02883=1217.618,361.256,-75.061,-175.943,7.642,148.283
C02884=1217.622,361.008,-75.028,-175.944,7.639,148.282
C02885=1217.626,360.760,-74.996,-175.945,7.636,148.282
C02886=1217.630,360.513,-74.963,-175.947,7.634,148.282
C02887=1217.634,360.265,-74.930,-175.949,7.630,148.282
C02888=1217.639,360.017,-74.897,-175.950,7.627,148.281
C02889=1217.643,359.769,-74.864,-175.952,7.625,148.281
C02890=1217.647,359.521,-74.831,-175.954,7.621,148.281
C02891=1217.650,359.274,-74.798,-175.955,7.619,148.280
C02892=1217.655,359.025,-74.766,-175.957,7.616,148.280
C02893=1217.659,358.778,-74.733,-175.959,7.613,148.280
C02894=1217.663,358.530,-74.700,-175.960,7.610,148.280
C02895=1217.667,358.283,-74.668,-175.962,7.607,148.279
C02896=1217.672,358.035,-74.635,-175.964,7.604,148.279
C02897=1217.676,357.787,-74.602,-175.965,7.601,148.279
C02898=1217.680,357.539,-74.569,-175.967,7.599,148.279
C02899=1217.684,357.291,-74.537,-175.969,7.595,148.278
C02900=1217.688,357.043,-74.504,-175.970,7.593,148.278
C02901=1217.692,356.795,-74.471,-175.972,7.590,148.278
C02902=1217.697,356.547,-74.439,-175.974,7.587,148.278
C02903=1217.700,356.300,-74.406,-175.975,7.584,148.277
C02904=1217.705,356.053,-74.373,-175.977,7.581,148.277
C02905=1217.709,355.804,-74.341,-175.979,7.578,148.277
C02906=1217.713,355.556,-74.308,-175.981,7.575,148.277
C02907=1217.717,355.308,-74.276,-175.982,7.573,148.276
C02908=1217.721,355.061,-74.243,-175.984,7.569,148.276
C02909=1217.726,354.812,-74.210,-175.986,7.567,148.276
C02910=1217.729,354.565,-74.178,-175.987,7.564,148.276
C02911=1217.734,354.317,-74.146,-175.989,7.561,148.275
C02912=1217.738,354.070,-74.112,-175.991,7.558,148.275
C02913=1217.742,353.821,-74.081,-175.992,7.556,148.275
C02914=1217.746,353.574,-74.047,-175.994,7.552,148.275
C02915=1217.750,353.325,-74.015,-175.996,7.550,148.274
C02916=1217.754,353.077,-73.983,-175.998,7.546,148.274
C02917=1217.759,352.830,-73.950,-176.000,7.544,148.274
C02918=1217.763,352.582,-73.918,-176.001,7.541,148.274
C02919=1217.767,352.335,-73.885,-176.003,7.538,148.273
C02920=1217.771,352.086,-73.853,-176.005,7.535,148.273
C02921=1217.775,351.838,-73.821,-176.007,7.533,148.273
C02922=1217.780,351.591,-73.788,-176.009,7.529,148.273
C02923=1217.784,351.343,-73.756,-176.010,7.527,148.273
C02924=1217.788,351.095,-73.724,-176.013,7.523,148.272
C02925=1217.792,350.847,-73.691,-176.014,7.521,148.272
C02926=1217.796,350.599,-73.659,-176.015,7.518,148.272
C02927=1217.801,350.351,-73.627,-176.018,7.515,148.271
C02928=1217.804,350.104,-73.594,-176.019,7.512,148.271
C02929=1217.809,349.856,-73.562,-176.021,7.510,148.271
C02930=1217.813,349.607,-73.530,-176.023,7.506,148.271
C02931=1217.817,349.360,-73.498,-176.025,7.504,148.271
C02932=1217.821,349.112,-73.465,-176.027,7.500,148.270
C02933=1217.825,348.864,-73.433,-176.029,7.498,148.270
C02934=1217.830,348.616,-73.401,-176.030,7.495,148.270
C02935=1217.834,348.368,-73.369,-176.032,7.492,148.270
C02936=1217.838,348.121,-73.336,-176.034,7.489,148.270
C02937=1217.842,347.873,-73.304,-176.036,7.486,148.269
C02938=1217.846,347.624,-73.272,-176.038,7.484,148.269
C02939=1217.850,347.377,-73.240,-176.040,7.481,148.269
C02940=1217.855,347.129,-73.208,-176.042,7.478,148.269
C02941=1217.859,346.881,-73.176,-176.043,7.475,148.269
C02942=1217.863,346.634,-73.143,-176.046,7.472,148.268
C02943=1217.867,346.386,-73.111,-176.047,7.469,148.268
C02944=1217.872,346.137,-73.079,-176.049,7.467,148.268
C02945=1217.875,345.889,-73.047,-176.051,7.463,148.268
C02946=1217.880,345.642,-73.016,-176.053,7.461,148.268
C02947=1217.884,345.393,-72.983,-176.055,7.458,148.268
C02948=1217.888,345.145,-72.951,-176.057,7.455,148.268
C02949=1217.893,344.898,-72.919,-176.059,7.452,148.267
C02950=1217.896,344.650,-72.887,-176.061,7.449,148.267
C02951=1217.901,344.401,-72.855,-176.062,7.447,148.267
C02952=1217.905,344.154,-72.823,-176.065,7.444,148.267
C02953=1217.909,343.906,-72.792,-176.066,7.441,148.267
C02954=1217.913,343.658,-72.759,-176.068,7.438,148.266
C02955=1217.918,343.410,-72.728,-176.070,7.435,148.266
C02956=1217.921,343.162,-72.696,-176.072,7.433,148.266
C02957=1217.926,342.914,-72.663,-176.074,7.430,148.266
C02958=1217.930,342.667,-72.632,-176.076,7.427,148.266
C02959=1217.935,342.418,-72.599,-176.078,7.424,148.266
C02960=1217.938,342.170,-72.568,-176.080,7.421,148.265
C02961=1217.943,341.923,-72.536,-176.082,7.418,148.265
C02962=1217.947,341.674,-72.504,-176.084,7.416,148.265
C02963=1217.951,341.397,-72.468,-176.086,7.412,148.265
C02964=1217.956,341.119,-72.432,-176.089,7.409,148.265
C02965=1217.961,340.841,-72.397,-176.091,7.406,148.264
C02966=1217.965,340.563,-72.361,-176.092,7.403,148.264
C02967=1217.970,340.315,-72.329,-176.095,7.400,148.264
C02968=1217.974,340.068,-72.297,-176.097,7.397,148.264
C02969=1217.978,339.819,-72.266,-176.099,7.394,148.264
C02970=1217.982,339.572,-72.235,-176.101,7.392,148.264
C02971=1217.987,339.323,-72.202,-176.103,7.389,148.264
C02972=1217.991,339.075,-72.171,-176.105,7.386,148.264
C02973=1217.995,338.828,-72.139,-176.107,7.384,148.263
C02974=1217.999,338.579,-72.108,-176.109,7.380,148.263
C02975=1218.003,338.332,-72.076,-176.111,7.378,148.263
C02976=1218.008,338.084,-72.044,-176.113,7.375,148.263
C02977=1218.011,337.836,-72.012,-176.115,7.372,148.263
C02978=1218.016,337.588,-71.981,-176.117,7.369,148.263
C02979=1218.020,337.340,-71.950,-176.119,7.367,148.263
C02980=1218.024,337.092,-71.918,-176.121,7.363,148.262
C02981=1218.028,336.844,-71.886,-176.123,7.361,148.262
C02982=1218.033,336.596,-71.855,-176.125,7.358,148.262
C02983=1218.037,336.348,-71.823,-176.127,7.355,148.262
C02984=1218.041,336.101,-71.792,-176.129,7.353,148.262
C02985=1218.045,335.852,-71.760,-176.131,7.349,148.262
C02986=1218.049,335.605,-71.729,-176.133,7.347,148.262
C02987=1218.054,335.356,-71.697,-176.136,7.344,148.262
C02988=1218.058,335.108,-71.665,-176.137,7.341,148.261
C02989=1218.062,334.860,-71.634,-176.140,7.338,148.261
C02990=1218.066,334.612,-71.602,-176.142,7.336,148.261
C02991=1218.070,334.364,-71.571,-176.143,7.333,148.261
C02992=1218.074,334.116,-71.539,-176.145,7.330,148.261
C02993=1218.079,333.868,-71.509,-176.148,7.328,148.261
C02994=1218.082,333.620,-71.477,-176.150,7.324,148.261
C02995=1218.087,333.372,-71.446,-176.152,7.322,148.261
C02996=1218.092,333.124,-71.414,-176.154,7.319,148.260
C02997=1218.096,332.876,-71.383,-176.156,7.317,148.261
C02998=1218.100,332.629,-71.351,-176.158,7.313,148.260
C02999=1218.104,332.380,-71.320,-176.160,7.311,148.260
C03000=1218.109,332.133,-71.289,-176.163,7.308,148.260
C03001=1218.113,331.884,-71.258,-176.164,7.305,148.260
C03002=1218.117,331.637,-71.226,-176.166,7.303,148.260
C03003=1218.121,331.388,-71.195,-176.169,7.300,148.260
C03004=1218.125,331.141,-71.164,-176.171,7.297,148.260
C03005=1218.129,330.892,-71.132,-176.173,7.294,148.260
C03006=1218.134,330.645,-71.101,-176.175,7.292,148.260
C03007=1218.138,330.396,-71.070,-176.177,7.288,148.259
C03008=1218.142,330.148,-71.039,-176.179,7.286,148.259
C03009=1218.147,329.901,-71.008,-176.182,7.283,148.259
C03010=1218.151,329.652,-70.976,-176.184,7.281,148.259
C03011=1218.155,329.405,-70.945,-176.186,7.277,148.259
C03012=1218.159,329.156,-70.914,-176.188,7.275,148.259
C03013=1218.164,328.908,-70.883,-176.190,7.273,148.259
C03014=1218.167,328.660,-70.851,-176.192,7.269,148.259
C03015=1218.172,328.412,-70.820,-176.194,7.267,148.259
C03016=1218.176,328.164,-70.790,-176.197,7.264,148.259
C03017=1218.180,327.916,-70.759,-176.198,7.261,148.259
C03018=1218.184,327.668,-70.728,-176.201,7.258,148.259
C03019=1218.188,327.420,-70.697,-176.202,7.256,148.258
C03020=1218.193,327.172,-70.666,-176.205,7.253,148.258
C03021=1218.197,326.924,-70.634,-176.207,7.251,148.258
C03022=1218.201,326.676,-70.603,-176.209,7.247,148.258
C03023=1218.206,326.428,-70.572,-176.212,7.245,148.258
C03024=1218.210,326.180,-70.542,-176.213,7.242,148.258
C03025=1218.214,325.932,-70.511,-176.216,7.239,148.258
C03026=1218.218,325.684,-70.480,-176.217,7.237,148.258
C03027=1218.222,325.436,-70.449,-176.220,7.234,148.258
C03028=1218.226,325.188,-70.418,-176.222,7.232,148.258
C03029=1218.231,324.940,-70.387,-176.224,7.228,148.258
C03030=1218.235,324.691,-70.356,-176.227,7.226,148.258
C03031=1218.239,324.443,-70.326,-176.229,7.223,148.258
C03032=1218.243,324.196,-70.294,-176.231,7.220,148.258
C03033=1218.247,323.947,-70.263,-176.234,7.217,148.258
C03034=1218.252,323.699,-70.232,-176.235,7.215,148.257
C03035=1218.257,323.451,-70.202,-176.237,7.213,148.257
C03036=1218.260,323.203,-70.171,-176.240,7.210,148.257
C03037=1218.264,322.955,-70.140,-176.242,7.207,148.257
C03038=1218.269,322.707,-70.109,-176.244,7.204,148.257
C03039=1218.274,322.459,-70.079,-176.246,7.202,148.257
C03040=1218.277,322.211,-70.048,-176.249,7.199,148.257
C03041=1218.282,321.963,-70.017,-176.251,7.196,148.257
C03042=1218.286,321.715,-69.987,-176.253,7.193,148.257
C03043=1218.289,321.467,-69.956,-176.255,7.191,148.257
C03044=1218.294,321.219,-69.925,-176.258,7.188,148.257
C03045=1218.299,320.971,-69.895,-176.260,7.185,148.257
C03046=1218.303,320.723,-69.864,-176.262,7.182,148.257
C03047=1218.307,320.474,-69.833,-176.264,7.180,148.257
C03048=1218.311,320.226,-69.803,-176.266,7.178,148.257
C03049=1218.316,319.978,-69.772,-176.269,7.175,148.257
C03050=1218.320,319.731,-69.742,-176.271,7.172,148.257
C03051=1218.324,319.482,-69.710,-176.273,7.169,148.257
C03052=1218.328,319.234,-69.680,-176.275,7.167,148.257
C03053=1218.332,318.986,-69.650,-176.278,7.164,148.257
C03054=1218.337,318.738,-69.619,-176.280,7.161,148.257
C03055=1218.341,318.489,-69.588,-176.282,7.158,148.257
C03056=1218.345,318.242,-69.558,-176.284,7.156,148.257
C03057=1218.350,317.994,-69.527,-176.287,7.153,148.257
C03058=1218.353,317.746,-69.497,-176.289,7.151,148.257
C03059=1218.358,317.497,-69.467,-176.291,7.148,148.257
C03060=1218.362,317.249,-69.436,-176.293,7.145,148.257
C03061=1218.366,317.001,-69.406,-176.296,7.143,148.257
C03062=1218.371,316.753,-69.375,-176.298,7.140,148.257
C03063=1218.375,316.506,-69.345,-176.300,7.138,148.257
C03064=1218.379,316.256,-69.315,-176.302,7.134,148.256
C03065=1218.383,316.009,-69.284,-176.305,7.132,148.256
C03066=1218.388,315.761,-69.254,-176.307,7.129,148.256
C03067=1218.393,315.484,-69.220,-176.309,7.127,148.257
C03068=1218.397,315.209,-69.186,-176.312,7.124,148.257
C03069=1218.402,314.932,-69.153,-176.315,7.121,148.257
C03070=1218.407,314.657,-69.119,-176.317,7.118,148.257
C03071=1218.410,314.409,-69.088,-176.319,7.115,148.256
C03072=1218.415,314.160,-69.058,-176.322,7.112,148.256
C03073=1218.419,313.913,-69.028,-176.324,7.110,148.256
C03074=1218.424,313.665,-68.997,-176.326,7.107,148.256
C03075=1218.428,313.417,-68.968,-176.329,7.105,148.256
C03076=1218.433,313.169,-68.937,-176.331,7.102,148.256
C03077=1218.436,312.920,-68.907,-176.333,7.099,148.257
C03078=1218.441,312.672,-68.877,-176.335,7.097,148.256
C03079=1218.445,312.423,-68.847,-176.338,7.094,148.256
C03080=1218.450,312.175,-68.816,-176.340,7.092,148.256
C03081=1218.453,311.928,-68.786,-176.342,7.089,148.256
C03082=1218.458,311.679,-68.757,-176.345,7.086,148.256
C03083=1218.462,311.432,-68.726,-176.347,7.083,148.256
C03084=1218.466,311.183,-68.697,-176.349,7.081,148.257
C03085=1218.471,310.935,-68.666,-176.352,7.078,148.257
C03086=1218.475,310.687,-68.636,-176.354,7.076,148.257
C03087=1218.479,310.439,-68.606,-176.356,7.074,148.257
C03088=1218.483,310.190,-68.576,-176.358,7.070,148.256
C03089=1218.487,309.942,-68.546,-176.361,7.068,148.256
C03090=1218.492,309.694,-68.516,-176.363,7.065,148.256
C03091=1218.496,309.446,-68.486,-176.365,7.063,148.257
C03092=1218.500,309.198,-68.456,-176.368,7.060,148.257
C03093=1218.505,308.949,-68.426,-176.370,7.058,148.257
C03094=1218.509,308.702,-68.396,-176.372,7.055,148.257
C03095=1218.513,308.453,-68.366,-176.375,7.052,148.257
C03096=1218.518,308.205,-68.336,-176.377,7.050,148.257
C03097=1218.522,307.957,-68.306,-176.380,7.047,148.257
C03098=1218.526,307.709,-68.277,-176.382,7.045,148.257
C03099=1218.531,307.460,-68.247,-176.384,7.042,148.257
C03100=1218.535,307.213,-68.216,-176.387,7.040,148.257
C03101=1218.539,306.964,-68.187,-176.389,7.037,148.257
C03102=1218.543,306.716,-68.157,-176.391,7.034,148.257
C03103=1218.548,306.468,-68.127,-176.393,7.032,148.257
C03104=1218.552,306.220,-68.097,-176.396,7.029,148.257
C03105=1218.556,305.972,-68.068,-176.398,7.027,148.257
C03106=1218.561,305.723,-68.038,-176.401,7.024,148.257
C03107=1218.565,305.475,-68.008,-176.403,7.022,148.257
C03108=1218.569,305.227,-67.978,-176.405,7.019,148.257
C03109=1218.574,304.979,-67.949,-176.408,7.016,148.257
C03110=1218.578,304.731,-67.919,-176.410,7.014,148.257
C03111=1218.583,304.482,-67.889,-176.413,7.011,148.257
C03112=1218.587,304.234,-67.859,-176.415,7.009,148.257
C03113=1218.591,303.986,-67.830,-176.417,7.006,148.257
C03114=1218.595,303.738,-67.800,-176.419,7.004,148.257
C03115=1218.600,303.489,-67.770,-176.422,7.001,148.257
C03116=1218.604,303.241,-67.741,-176.424,6.998,148.257
C03117=1218.608,302.993,-67.711,-176.426,6.996,148.257
C03118=1218.612,302.745,-67.682,-176.429,6.993,148.257
C03119=1218.616,302.497,-67.651,-176.431,6.991,148.258
C03120=1218.620,302.249,-67.622,-176.433,6.989,148.258
C03121=1218.625,302.001,-67.593,-176.436,6.986,148.258
C03122=1218.630,301.752,-67.563,-176.438,6.984,148.258
C03123=1218.634,301.504,-67.533,-176.441,6.981,148.258
C03124=1218.638,301.256,-67.504,-176.443,6.979,148.258
C03125=1218.643,301.008,-67.475,-176.445,6.976,148.258
C03126=1218.647,300.759,-67.445,-176.448,6.973,148.258
C03127=1218.651,300.511,-67.416,-176.450,6.971,148.258
C03128=1218.655,300.263,-67.386,-176.453,6.968,148.258
C03129=1218.659,300.015,-67.357,-176.455,6.966,148.258
C03130=1218.664,299.766,-67.327,-176.457,6.964,148.258
C03131=1218.668,299.519,-67.298,-176.460,6.961,148.258
C03132=1218.673,299.271,-67.269,-176.462,6.958,148.258
C03133=1218.677,299.022,-67.239,-176.465,6.956,148.258
C03134=1218.681,298.774,-67.210,-176.467,6.953,148.259
C03135=1218.686,298.525,-67.180,-176.469,6.951,148.259
C03136=1218.690,298.277,-67.151,-176.472,6.948,148.259
C03137=1218.694,298.028,-67.122,-176.474,6.946,148.259
C03138=1218.699,297.780,-67.092,-176.477,6.943,148.259
C03139=1218.703,297.532,-67.063,-176.479,6.941,148.259
C03140=1218.708,297.284,-67.034,-176.481,6.939,148.259
C03141=1218.711,297.036,-67.005,-176.484,6.936,148.259
C03142=1218.715,296.788,-66.975,-176.486,6.934,148.259
C03143=1218.720,296.539,-66.947,-176.489,6.931,148.259
C03144=1218.724,296.291,-66.917,-176.491,6.928,148.259
C03145=1218.729,296.043,-66.888,-176.493,6.926,148.259
C03146=1218.733,295.795,-66.859,-176.496,6.923,148.259
C03147=1218.737,295.547,-66.829,-176.498,6.921,148.260
C03148=1218.742,295.298,-66.800,-176.501,6.919,148.260
C03149=1218.746,295.050,-66.771,-176.503,6.916,148.260
C03150=1218.751,294.802,-66.742,-176.505,6.914,148.260
C03151=1218.755,294.554,-66.712,-176.508,6.911,148.260
C03152=1218.759,294.305,-66.684,-176.510,6.909,148.260
C03153=1218.763,294.057,-66.654,-176.513,6.907,148.260
C03154=1218.767,293.809,-66.625,-176.515,6.904,148.260
C03155=1218.772,293.560,-66.597,-176.517,6.901,148.260
C03156=1218.776,293.312,-66.567,-176.520,6.899,148.260
C03157=1218.780,293.064,-66.538,-176.522,6.896,148.260
C03158=1218.785,292.815,-66.509,-176.525,6.894,148.260
C03159=1218.790,292.567,-66.480,-176.528,6.891,148.260
C03160=1218.794,292.319,-66.451,-176.530,6.889,148.261
C03161=1218.797,292.071,-66.423,-176.532,6.887,148.261
C03162=1218.802,291.822,-66.393,-176.535,6.884,148.261
C03163=1218.807,291.574,-66.365,-176.537,6.882,148.261
C03164=1218.811,291.326,-66.335,-176.539,6.880,148.261
C03165=1218.815,291.077,-66.307,-176.542,6.877,148.261
C03166=1218.819,290.829,-66.278,-176.544,6.874,148.261
C03167=1218.824,290.581,-66.249,-176.547,6.872,148.261
C03168=1218.828,290.333,-66.220,-176.549,6.869,148.261
C03169=1218.832,290.084,-66.190,-176.551,6.867,148.261
C03170=1218.837,289.836,-66.162,-176.554,6.864,148.261
C03171=1218.842,289.562,-66.130,-176.557,6.862,148.262
C03172=1218.847,289.288,-66.098,-176.559,6.859,148.262
C03173=1218.851,289.014,-66.066,-176.562,6.857,148.262
C03174=1218.856,288.739,-66.035,-176.565,6.854,148.262
C03175=1218.860,288.491,-66.006,-176.567,6.851,148.262
C03176=1218.865,288.243,-65.978,-176.570,6.849,148.262
C03177=1218.869,287.994,-65.949,-176.572,6.847,148.262
C03178=1218.873,287.746,-65.920,-176.575,6.844,148.262
C03179=1218.878,287.498,-65.892,-176.577,6.842,148.262
C03180=1218.882,287.250,-65.862,-176.579,6.840,148.263
C03181=1218.887,287.001,-65.833,-176.582,6.837,148.263
C03182=1218.891,286.753,-65.806,-176.584,6.835,148.263
C03183=1218.895,286.505,-65.776,-176.587,6.833,148.263
C03184=1218.899,286.256,-65.748,-176.589,6.830,148.263
C03185=1218.904,286.008,-65.720,-176.592,6.828,148.263
C03186=1218.908,285.760,-65.690,-176.594,6.826,148.264
C03187=1218.912,285.511,-65.662,-176.597,6.823,148.264
C03188=1218.917,285.263,-65.634,-176.599,6.821,148.264
C03189=1218.921,285.014,-65.605,-176.601,6.818,148.264
C03190=1218.925,284.767,-65.576,-176.604,6.816,148.264
C03191=1218.930,284.518,-65.548,-176.606,6.813,148.264
C03192=1218.934,284.269,-65.520,-176.608,6.811,148.264
C03193=1218.939,284.021,-65.491,-176.612,6.808,148.264
C03194=1218.943,283.773,-65.462,-176.614,6.806,148.264
C03195=1218.947,283.525,-65.434,-176.616,6.804,148.264
C03196=1218.952,283.276,-65.405,-176.619,6.801,148.265
C03197=1218.956,283.028,-65.377,-176.621,6.799,148.265
C03198=1218.961,282.779,-65.349,-176.623,6.797,148.265
C03199=1218.964,282.531,-65.321,-176.626,6.794,148.265
C03200=1218.969,282.283,-65.292,-176.629,6.792,148.265
C03201=1218.973,282.035,-65.263,-176.631,6.790,148.265
C03202=1218.978,281.787,-65.235,-176.634,6.787,148.265
C03203=1218.982,281.538,-65.207,-176.636,6.785,148.265
C03204=1218.987,281.290,-65.178,-176.639,6.783,148.266
C03205=1218.991,281.041,-65.150,-176.641,6.781,148.266
C03206=1218.996,280.793,-65.122,-176.643,6.778,148.266
C03207=1218.999,280.544,-65.094,-176.646,6.776,148.266
C03208=1219.004,280.296,-65.065,-176.648,6.774,148.266
C03209=1219.008,280.048,-65.037,-176.651,6.771,148.266
C03210=1219.013,279.799,-65.009,-176.653,6.769,148.267
C03211=1219.017,279.551,-64.981,-176.655,6.767,148.267
C03212=1219.022,279.302,-64.952,-176.659,6.764,148.267
C03213=1219.026,279.054,-64.924,-176.661,6.762,148.267
C03214=1219.030,278.806,-64.896,-176.663,6.759,148.267
C03215=1219.035,278.557,-64.868,-176.665,6.758,148.267
C03216=1219.039,278.309,-64.840,-176.668,6.754,148.267
C03217=1219.044,278.061,-64.811,-176.671,6.753,148.268
C03218=1219.047,277.812,-64.783,-176.673,6.750,148.268
C03219=1219.052,277.564,-64.755,-176.676,6.747,148.268
C03220=1219.056,277.315,-64.727,-176.678,6.745,148.268
C03221=1219.061,277.067,-64.699,-176.680,6.743,148.268
C03222=1219.066,276.819,-64.670,-176.683,6.741,148.268
C03223=1219.069,276.571,-64.642,-176.686,6.738,148.268
C03224=1219.074,276.323,-64.615,-176.688,6.736,148.269
C03225=1219.078,276.074,-64.586,-176.690,6.734,148.269
C03226=1219.083,275.825,-64.559,-176.693,6.731,148.269
C03227=1219.087,275.577,-64.531,-176.696,6.729,148.269
C03228=1219.092,275.329,-64.502,-176.698,6.727,148.269
C03229=1219.095,275.080,-64.474,-176.700,6.725,148.269
C03230=1219.100,274.832,-64.446,-176.703,6.722,148.269
C03231=1219.104,274.584,-64.419,-176.706,6.720,148.270
C03232=1219.109,274.335,-64.390,-176.708,6.718,148.270
C03233=1219.113,274.087,-64.363,-176.710,6.716,148.270
C03234=1219.117,273.838,-64.335,-176.713,6.713,148.270
C03235=1219.122,273.589,-64.307,-176.715,6.711,148.270
C03236=1219.127,273.342,-64.279,-176.718,6.709,148.271
C03237=1219.131,273.093,-64.251,-176.720,6.707,148.271
C03238=1219.135,272.845,-64.223,-176.723,6.704,148.271
C03239=1219.140,272.596,-64.195,-176.725,6.702,148.271
C03240=1219.144,272.348,-64.167,-176.728,6.700,148.271
C03241=1219.148,272.100,-64.140,-176.730,6.698,148.271
C03242=1219.152,271.851,-64.112,-176.733,6.695,148.272
C03243=1219.157,271.603,-64.084,-176.735,6.693,148.272
C03244=1219.162,271.355,-64.056,-176.738,6.691,148.272
C03245=1219.166,271.105,-64.029,-176.740,6.689,148.272
C03246=1219.170,270.858,-64.001,-176.743,6.686,148.272
C03247=1219.174,270.608,-63.973,-176.745,6.684,148.272
C03248=1219.179,270.361,-63.946,-176.748,6.682,148.273
C03249=1219.183,270.113,-63.918,-176.750,6.680,148.273
C03250=1219.188,269.863,-63.890,-176.753,6.677,148.273
C03251=1219.192,269.615,-63.862,-176.755,6.675,148.273
C03252=1219.197,269.367,-63.835,-176.758,6.673,148.273
C03253=1219.201,269.118,-63.807,-176.760,6.671,148.273
C03254=1219.205,268.870,-63.780,-176.763,6.668,148.274
C03255=1219.210,268.622,-63.752,-176.765,6.666,148.274
C03256=1219.214,268.373,-63.725,-176.768,6.664,148.274
C03257=1219.218,268.125,-63.697,-176.770,6.662,148.274
C03258=1219.223,267.876,-63.669,-176.773,6.660,148.274
C03259=1219.228,267.628,-63.641,-176.775,6.657,148.274
C03260=1219.232,267.379,-63.614,-176.778,6.655,148.275
C03261=1219.236,267.131,-63.586,-176.780,6.653,148.275
C03262=1219.241,266.882,-63.559,-176.783,6.651,148.275
C03263=1219.245,266.634,-63.532,-176.785,6.648,148.275
C03264=1219.249,266.385,-63.504,-176.788,6.646,148.275
C03265=1219.254,266.137,-63.477,-176.790,6.644,148.276
C03266=1219.258,265.889,-63.449,-176.793,6.642,148.276
C03267=1219.263,265.641,-63.422,-176.795,6.640,148.276
C03268=1219.267,265.391,-63.395,-176.798,6.637,148.276
C03269=1219.271,265.143,-63.367,-176.800,6.635,148.276
C03270=1219.276,264.895,-63.340,-176.803,6.633,148.277
C03271=1219.281,264.646,-63.313,-176.805,6.631,148.277
C03272=1219.284,264.398,-63.285,-176.807,6.629,148.277
C03273=1219.289,264.149,-63.257,-176.810,6.626,148.277
C03274=1219.294,263.901,-63.230,-176.813,6.624,148.277
C03275=1219.299,263.628,-63.200,-176.815,6.622,148.278
C03276=1219.303,263.356,-63.170,-176.818,6.620,148.278
C03277=1219.307,263.083,-63.140,-176.821,6.617,148.278
C03278=1219.313,262.810,-63.110,-176.824,6.615,148.278
C03279=1219.317,262.562,-63.083,-176.826,6.613,148.278
C03280=1219.322,262.313,-63.056,-176.828,6.611,148.279
C03281=1219.327,262.065,-63.029,-176.831,6.609,148.279
C03282=1219.331,261.816,-63.001,-176.834,6.606,148.279
C03283=1219.335,261.568,-62.974,-176.836,6.604,148.279
C03284=1219.339,261.320,-62.947,-176.838,6.602,148.279
C03285=1219.344,261.071,-62.920,-176.841,6.600,148.280
C03286=1219.348,260.823,-62.893,-176.844,6.598,148.280
C03287=1219.353,260.574,-62.866,-176.846,6.596,148.280
C03288=1219.357,260.325,-62.839,-176.849,6.593,148.280
C03289=1219.361,260.077,-62.811,-176.851,6.591,148.280
C03290=1219.366,259.829,-62.784,-176.854,6.589,148.281
C03291=1219.370,259.580,-62.757,-176.856,6.587,148.281
C03292=1219.375,259.332,-62.730,-176.858,6.585,148.281
C03293=1219.379,259.083,-62.703,-176.862,6.582,148.281
C03294=1219.384,258.835,-62.676,-176.864,6.580,148.281
C03295=1219.388,258.586,-62.649,-176.866,6.578,148.282
C03296=1219.393,258.337,-62.622,-176.869,6.576,148.282
C03297=1219.397,258.089,-62.595,-176.871,6.574,148.282
C03298=1219.401,257.841,-62.568,-176.874,6.572,148.282
C03299=1219.406,257.592,-62.541,-176.876,6.570,148.282
C03300=1219.410,257.344,-62.514,-176.879,6.567,148.283
C03301=1219.414,257.095,-62.487,-176.882,6.565,148.283
C03302=1219.419,256.847,-62.460,-176.884,6.563,148.283
C03303=1219.424,256.598,-62.433,-176.886,6.561,148.283
C03304=1219.428,256.350,-62.406,-176.889,6.559,148.284
C03305=1219.432,256.101,-62.379,-176.891,6.557,148.284
C03306=1219.436,255.852,-62.352,-176.894,6.554,148.284
C03307=1219.441,255.604,-62.325,-176.896,6.552,148.284
C03308=1219.446,255.355,-62.298,-176.899,6.550,148.284
C03309=1219.450,255.107,-62.273,-176.902,6.548,148.285
C03310=1219.455,254.858,-62.245,-176.904,6.546,148.285
C03311=1219.459,254.610,-62.218,-176.906,6.544,148.285
C03312=1219.463,254.361,-62.192,-176.909,6.542,148.285
C03313=1219.468,254.113,-62.165,-176.912,6.539,148.285
C03314=1219.472,253.865,-62.138,-176.914,6.538,148.286
C03315=1219.476,253.616,-62.111,-176.917,6.536,148.286
C03316=1219.481,253.367,-62.085,-176.919,6.534,148.286
C03317=1219.486,253.119,-62.058,-176.922,6.532,148.286
C03318=1219.490,252.871,-62.031,-176.924,6.530,148.287
C03319=1219.495,252.622,-62.004,-176.926,6.528,148.287
C03320=1219.500,252.373,-61.978,-176.929,6.526,148.287
C03321=1219.503,252.125,-61.952,-176.932,6.523,148.287
C03322=1219.508,251.876,-61.925,-176.934,6.521,148.288
C03323=1219.512,251.628,-61.898,-176.937,6.519,148.288
C03324=1219.517,251.379,-61.872,-176.940,6.517,148.288
C03325=1219.522,251.130,-61.845,-176.942,6.515,148.288
C03326=1219.526,250.882,-61.818,-176.944,6.513,148.289
C03327=1219.530,250.634,-61.791,-176.947,6.511,148.289
C03328=1219.534,250.385,-61.765,-176.949,6.509,148.289
C03329=1219.539,250.136,-61.738,-176.952,6.507,148.289
C03330=1219.543,249.888,-61.712,-176.955,6.504,148.290
C03331=1219.548,249.639,-61.685,-176.957,6.502,148.290
C03332=1219.552,249.391,-61.659,-176.960,6.500,148.290
C03333=1219.557,249.142,-61.633,-176.962,6.498,148.290
C03334=1219.561,248.894,-61.606,-176.964,6.496,148.290
C03335=1219.565,248.645,-61.579,-176.967,6.494,148.291
C03336=1219.570,248.396,-61.553,-176.970,6.492,148.291
C03337=1219.574,248.148,-61.526,-176.972,6.491,148.291
C03338=1219.579,247.899,-61.501,-176.974,6.488,148.291
C03339=1219.583,247.651,-61.474,-176.977,6.487,148.292
C03340=1219.587,247.402,-61.448,-176.980,6.484,148.292
C03341=1219.592,247.153,-61.421,-176.982,6.482,148.292
C03342=1219.597,246.905,-61.395,-176.985,6.480,148.292
C03343=1219.602,246.657,-61.368,-176.987,6.478,148.293
C03344=1219.606,246.408,-61.343,-176.990,6.476,148.293
C03345=1219.610,246.159,-61.315,-176.992,6.474,148.293
C03346=1219.615,245.911,-61.290,-176.995,6.472,148.293
C03347=1219.619,245.662,-61.263,-176.997,6.470,148.294
C03348=1219.624,245.413,-61.237,-177.000,6.468,148.294
C03349=1219.627,245.165,-61.210,-177.002,6.466,148.294
C03350=1219.632,244.916,-61.184,-177.005,6.464,148.294
C03351=1219.637,244.668,-61.158,-177.007,6.462,148.295
C03352=1219.642,244.419,-61.132,-177.010,6.459,148.295
C03353=1219.646,244.171,-61.106,-177.013,6.457,148.295
C03354=1219.650,243.922,-61.079,-177.015,6.456,148.295
C03355=1219.655,243.673,-61.053,-177.018,6.453,148.295
C03356=1219.659,243.425,-61.027,-177.020,6.451,148.296
C03357=1219.663,243.176,-61.001,-177.023,6.450,148.296
C03358=1219.669,242.928,-60.975,-177.025,6.448,148.296
C03359=1219.673,242.680,-60.948,-177.028,6.446,148.296
C03360=1219.677,242.431,-60.923,-177.030,6.444,148.297
C03361=1219.682,242.182,-60.896,-177.033,6.442,148.297
C03362=1219.686,241.933,-60.871,-177.035,6.440,148.297
C03363=1219.690,241.685,-60.844,-177.038,6.438,148.298
C03364=1219.696,241.436,-60.818,-177.040,6.436,148.298
C03365=1219.700,241.188,-60.792,-177.043,6.434,148.298
C03366=1219.704,240.939,-60.767,-177.045,6.432,148.298
C03367=1219.708,240.691,-60.740,-177.048,6.429,148.299
C03368=1219.713,240.441,-60.714,-177.051,6.427,148.299
C03369=1219.718,240.193,-60.688,-177.053,6.425,148.299
C03370=1219.722,239.945,-60.663,-177.056,6.424,148.299
C03371=1219.726,239.696,-60.636,-177.059,6.422,148.300
C03372=1219.731,239.447,-60.610,-177.061,6.420,148.300
C03373=1219.735,239.198,-60.584,-177.063,6.418,148.300
C03374=1219.740,238.950,-60.559,-177.066,6.416,148.300
C03375=1219.744,238.702,-60.533,-177.069,6.414,148.301
C03376=1219.749,238.452,-60.507,-177.071,6.412,148.301
C03377=1219.753,238.204,-60.480,-177.073,6.410,148.301
C03378=1219.758,237.956,-60.455,-177.076,6.408,148.302
C03379=1219.762,237.684,-60.427,-177.079,6.406,148.302
C03380=1219.767,237.412,-60.399,-177.082,6.403,148.302
C03381=1219.772,237.142,-60.370,-177.084,6.402,148.302
C03382=1219.777,236.870,-60.342,-177.087,6.400,148.303
C03383=1219.782,236.622,-60.317,-177.090,6.398,148.303
C03384=1219.787,236.373,-60.291,-177.092,6.396,148.303
C03385=1219.791,236.124,-60.265,-177.094,6.394,148.304
C03386=1219.795,235.875,-60.239,-177.097,6.392,148.304
C03387=1219.800,235.627,-60.214,-177.100,6.390,148.304
C03388=1219.804,235.378,-60.188,-177.102,6.388,148.304
C03389=1219.808,235.129,-60.162,-177.104,6.386,148.305
C03390=1219.813,234.881,-60.137,-177.107,6.384,148.305
C03391=1219.817,234.632,-60.111,-177.110,6.382,148.305
C03392=1219.822,234.383,-60.085,-177.112,6.380,148.306
C03393=1219.827,234.135,-60.059,-177.115,6.379,148.306
C03394=1219.831,233.886,-60.034,-177.118,6.376,148.306
C03395=1219.836,233.638,-60.008,-177.120,6.374,148.306
C03396=1219.840,233.389,-59.982,-177.123,6.372,148.307
C03397=1219.845,233.141,-59.957,-177.125,6.370,148.307
C03398=1219.849,232.892,-59.931,-177.128,6.368,148.307
C03399=1219.854,232.643,-59.906,-177.131,6.366,148.307
C03400=1219.858,232.394,-59.880,-177.133,6.364,148.308
C03401=1219.862,232.146,-59.855,-177.135,6.362,148.308
C03402=1219.867,231.897,-59.829,-177.138,6.360,148.308
C03403=1219.872,231.649,-59.804,-177.141,6.358,148.309
C03404=1219.876,231.400,-59.778,-177.143,6.357,148.309
C03405=1219.881,231.152,-59.752,-177.146,6.355,148.309
C03406=1219.885,230.902,-59.727,-177.148,6.353,148.309
C03407=1219.889,230.653,-59.702,-177.151,6.351,148.310
C03408=1219.894,230.405,-59.676,-177.153,6.349,148.310
C03409=1219.898,230.157,-59.651,-177.156,6.347,148.310
C03410=1219.904,229.908,-59.626,-177.159,6.345,148.311
C03411=1219.908,229.659,-59.600,-177.161,6.343,148.311
C03412=1219.912,229.410,-59.574,-177.163,6.341,148.311
C03413=1219.917,229.162,-59.549,-177.166,6.339,148.311
C03414=1219.921,228.913,-59.524,-177.169,6.337,148.312
C03415=1219.926,228.665,-59.499,-177.171,6.335,148.312
C03416=1219.930,228.416,-59.473,-177.174,6.334,148.312
C03417=1219.934,228.167,-59.448,-177.176,6.333,148.313
C03418=1219.939,227.919,-59.423,-177.179,6.331,148.313
C03419=1219.943,227.670,-59.397,-177.181,6.329,148.313
C03420=1219.948,227.421,-59.373,-177.183,6.327,148.313
C03421=1219.953,227.172,-59.347,-177.186,6.325,148.314
C03422=1219.957,226.924,-59.321,-177.189,6.323,148.314
C03423=1219.962,226.675,-59.296,-177.191,6.321,148.314
C03424=1219.966,226.427,-59.272,-177.194,6.319,148.315
C03425=1219.971,226.177,-59.247,-177.196,6.317,148.315
C03426=1219.975,225.929,-59.221,-177.199,6.316,148.315
C03427=1219.980,225.681,-59.195,-177.201,6.313,148.315
C03428=1219.984,225.431,-59.170,-177.204,6.311,148.316
C03429=1219.989,225.183,-59.145,-177.207,6.310,148.316
C03430=1219.993,224.934,-59.121,-177.209,6.308,148.316
C03431=1219.998,224.686,-59.095,-177.212,6.306,148.317
C03432=1220.002,224.436,-59.070,-177.214,6.304,148.317
C03433=1220.007,224.188,-59.045,-177.217,6.302,148.317
C03434=1220.011,223.939,-59.020,-177.220,6.300,148.318
C03435=1220.016,223.691,-58.995,-177.222,6.298,148.318
C03436=1220.020,223.442,-58.970,-177.225,6.297,148.318
C03437=1220.025,223.194,-58.945,-177.227,6.294,148.318
C03438=1220.029,222.944,-58.919,-177.230,6.293,148.319
C03439=1220.034,222.696,-58.895,-177.232,6.291,148.319
C03440=1220.038,222.447,-58.870,-177.235,6.289,148.319
C03441=1220.043,222.199,-58.844,-177.238,6.287,148.320
C03442=1220.048,221.950,-58.820,-177.240,6.285,148.320
C03443=1220.052,221.701,-58.795,-177.243,6.283,148.320
C03444=1220.057,221.453,-58.770,-177.245,6.281,148.321
C03445=1220.061,221.203,-58.745,-177.248,6.280,148.321
C03446=1220.066,220.955,-58.721,-177.251,6.278,148.321
C03447=1220.070,220.706,-58.695,-177.253,6.276,148.322
C03448=1220.075,220.458,-58.670,-177.255,6.275,148.322
C03449=1220.079,220.208,-58.646,-177.258,6.273,148.322
C03450=1220.084,219.960,-58.620,-177.260,6.271,148.323
C03451=1220.089,219.712,-58.596,-177.263,6.269,148.323
C03452=1220.092,219.462,-58.571,-177.265,6.267,148.323
C03453=1220.097,219.214,-58.546,-177.268,6.265,148.324
C03454=1220.102,218.965,-58.521,-177.271,6.263,148.324
C03455=1220.106,218.717,-58.497,-177.273,6.262,148.324
C03456=1220.111,218.467,-58.472,-177.276,6.260,148.325
C03457=1220.116,218.219,-58.446,-177.279,6.258,148.325
C03458=1220.120,217.971,-58.422,-177.281,6.256,148.325
C03459=1220.124,217.721,-58.397,-177.284,6.254,148.326
C03460=1220.129,217.473,-58.373,-177.287,6.252,148.326
C03461=1220.133,217.224,-58.347,-177.289,6.250,148.326
C03462=1220.138,216.975,-58.323,-177.292,6.249,148.327
C03463=1220.143,216.727,-58.299,-177.294,6.247,148.327
C03464=1220.147,216.477,-58.274,-177.297,6.245,148.327
C03465=1220.152,216.229,-58.250,-177.300,6.243,148.328
C03466=1220.157,215.980,-58.225,-177.302,6.242,148.328
C03467=1220.160,215.732,-58.200,-177.304,6.240,148.328
C03468=1220.165,215.483,-58.175,-177.307,6.238,148.328
C03469=1220.170,215.235,-58.151,-177.309,6.236,148.329
C03470=1220.174,214.985,-58.126,-177.312,6.234,148.329
C03471=1220.179,214.737,-58.102,-177.314,6.232,148.329
C03472=1220.184,214.488,-58.077,-177.317,6.231,148.330
C03473=1220.188,214.239,-58.053,-177.320,6.229,148.330
C03474=1220.193,213.990,-58.028,-177.322,6.227,148.330
C03475=1220.197,213.742,-58.004,-177.325,6.225,148.331
C03476=1220.202,213.492,-57.979,-177.328,6.223,148.331
C03477=1220.206,213.244,-57.955,-177.330,6.221,148.331
C03478=1220.211,212.995,-57.930,-177.333,6.219,148.332
C03479=1220.215,212.746,-57.906,-177.335,6.218,148.332
C03480=1220.220,212.497,-57.881,-177.338,6.217,148.332
C03481=1220.224,212.249,-57.857,-177.340,6.215,148.333
C03482=1220.230,212.000,-57.832,-177.343,6.213,148.333
C03483=1220.233,211.730,-57.806,-177.346,6.211,148.333
C03484=1220.239,211.460,-57.779,-177.349,6.209,148.334
C03485=1220.244,211.189,-57.753,-177.352,6.207,148.334
C03486=1220.249,210.919,-57.727,-177.354,6.205,148.335
C03487=1220.253,210.669,-57.702,-177.357,6.203,148.335
C03488=1220.258,210.421,-57.677,-177.360,6.201,148.335
C03489=1220.262,210.172,-57.653,-177.362,6.199,148.336
C03490=1220.267,209.924,-57.629,-177.364,6.198,148.336
C03491=1220.271,209.674,-57.604,-177.367,6.197,148.336
C03492=1220.276,209.426,-57.580,-177.370,6.195,148.337
C03493=1220.280,209.178,-57.556,-177.372,6.193,148.337
C03494=1220.286,208.928,-57.532,-177.375,6.191,148.337
C03495=1220.290,208.680,-57.508,-177.378,6.189,148.338
C03496=1220.294,208.431,-57.484,-177.380,6.187,148.338
C03497=1220.299,208.182,-57.459,-177.383,6.185,148.338
C03498=1220.303,207.934,-57.435,-177.385,6.184,148.339
C03499=1220.308,207.685,-57.412,-177.388,6.183,148.339
C03500=1220.313,207.436,-57.387,-177.390,6.181,148.339
C03501=1220.317,207.187,-57.362,-177.393,6.179,148.340
C03502=1220.321,206.938,-57.338,-177.396,6.177,148.340
C03503=1220.327,206.689,-57.314,-177.398,6.175,148.340
C03504=1220.331,206.441,-57.290,-177.401,6.173,148.341
C03505=1220.336,206.192,-57.266,-177.403,6.172,148.341
C03506=1220.339,205.943,-57.242,-177.406,6.171,148.341
C03507=1220.345,205.694,-57.218,-177.408,6.169,148.342
C03508=1220.349,205.445,-57.194,-177.411,6.167,148.342
C03509=1220.354,205.197,-57.170,-177.413,6.165,148.342
C03510=1220.358,204.948,-57.146,-177.416,6.163,148.343
C03511=1220.363,204.699,-57.122,-177.419,6.161,148.343
C03512=1220.367,204.450,-57.097,-177.421,6.159,148.343
C03513=1220.372,204.201,-57.074,-177.424,6.158,148.344
C03514=1220.376,203.953,-57.050,-177.426,6.157,148.344
C03515=1220.381,203.704,-57.026,-177.429,6.155,148.344
C03516=1220.386,203.455,-57.002,-177.432,6.153,148.345
C03517=1220.391,203.206,-56.978,-177.434,6.151,148.345
C03518=1220.395,202.957,-56.954,-177.437,6.150,148.346
C03519=1220.399,202.708,-56.930,-177.440,6.148,148.346
C03520=1220.404,202.459,-56.907,-177.442,6.147,148.346
C03521=1220.408,202.211,-56.882,-177.444,6.145,148.347
C03522=1220.413,201.962,-56.858,-177.447,6.143,148.347
C03523=1220.418,201.713,-56.834,-177.450,6.141,148.347
C03524=1220.422,201.465,-56.810,-177.452,6.139,148.348
C03525=1220.427,201.216,-56.787,-177.455,6.137,148.348
C03526=1220.431,200.967,-56.763,-177.457,6.136,148.348
C03527=1220.436,200.718,-56.740,-177.460,6.135,148.349
C03528=1220.441,200.470,-56.715,-177.462,6.133,148.349
C03529=1220.445,200.221,-56.692,-177.465,6.131,148.350
C03530=1220.449,199.971,-56.668,-177.468,6.129,148.350
C03531=1220.454,199.723,-56.644,-177.470,6.127,148.350
C03532=1220.459,199.473,-56.620,-177.472,6.126,148.351
C03533=1220.464,199.225,-56.596,-177.475,6.124,148.351
C03534=1220.468,198.976,-56.573,-177.478,6.123,148.351
C03535=1220.473,198.727,-56.549,-177.481,6.121,148.352
C03536=1220.477,198.478,-56.525,-177.483,6.119,148.352
C03537=1220.482,198.229,-56.502,-177.486,6.117,148.352
C03538=1220.486,197.981,-56.478,-177.488,6.116,148.353
C03539=1220.491,197.732,-56.455,-177.491,6.115,148.353
C03540=1220.496,197.483,-56.431,-177.494,6.113,148.354
C03541=1220.500,197.234,-56.407,-177.496,6.111,148.354
C03542=1220.505,196.985,-56.384,-177.499,6.109,148.354
C03543=1220.510,196.736,-56.361,-177.501,6.108,148.355
C03544=1220.514,196.488,-56.336,-177.504,6.106,148.355
C03545=1220.519,196.239,-56.313,-177.506,6.104,148.355
C03546=1220.523,195.990,-56.290,-177.509,6.103,148.356
C03547=1220.528,195.742,-56.266,-177.512,6.101,148.356
C03548=1220.533,195.492,-56.242,-177.514,6.100,148.357
C03549=1220.537,195.243,-56.219,-177.517,6.098,148.357
C03550=1220.542,194.994,-56.196,-177.519,6.096,148.357
C03551=1220.546,194.746,-56.172,-177.522,6.094,148.358
C03552=1220.550,194.497,-56.149,-177.525,6.093,148.358
C03553=1220.555,194.248,-56.125,-177.527,6.092,148.358
C03554=1220.560,193.999,-56.102,-177.529,6.090,148.359
C03555=1220.564,193.750,-56.079,-177.532,6.088,148.359
C03556=1220.569,193.502,-56.055,-177.535,6.086,148.360
C03557=1220.573,193.253,-56.031,-177.538,6.085,148.360
C03558=1220.578,193.004,-56.008,-177.540,6.084,148.360
C03559=1220.583,192.755,-55.985,-177.542,6.082,148.361
C03560=1220.588,192.506,-55.961,-177.545,6.080,148.361
C03561=1220.592,192.257,-55.938,-177.548,6.078,148.361
C03562=1220.597,192.009,-55.915,-177.550,6.077,148.362
C03563=1220.601,191.760,-55.891,-177.553,6.075,148.362
C03564=1220.606,191.511,-55.868,-177.555,6.073,148.362
C03565=1220.611,191.262,-55.845,-177.558,6.072,148.363
C03566=1220.615,191.013,-55.821,-177.561,6.070,148.363
C03567=1220.620,190.764,-55.798,-177.563,6.069,148.364
C03568=1220.624,190.515,-55.775,-177.566,6.067,148.364
C03569=1220.629,190.266,-55.752,-177.568,6.065,148.364
C03570=1220.633,190.017,-55.728,-177.571,6.063,148.365
C03571=1220.638,189.768,-55.705,-177.573,6.062,148.365
C03572=1220.643,189.520,-55.682,-177.576,6.061,148.366
C03573=1220.648,189.271,-55.659,-177.579,6.059,148.366
C03574=1220.652,189.022,-55.636,-177.581,6.057,148.366
C03575=1220.657,188.773,-55.613,-177.584,6.056,148.367
C03576=1220.661,188.524,-55.589,-177.586,6.054,148.367
C03577=1220.666,188.275,-55.566,-177.589,6.053,148.368
C03578=1220.670,188.026,-55.543,-177.592,6.051,148.368
C03579=1220.675,187.777,-55.520,-177.594,6.050,148.368
C03580=1220.680,187.529,-55.497,-177.597,6.048,148.369
C03581=1220.685,187.280,-55.473,-177.599,6.046,148.369
C03582=1220.689,187.031,-55.451,-177.602,6.045,148.370
C03583=1220.694,186.782,-55.428,-177.604,6.044,148.370
C03584=1220.699,186.533,-55.405,-177.607,6.042,148.370
C03585=1220.702,186.284,-55.382,-177.609,6.040,148.371
C03586=1220.708,186.035,-55.359,-177.612,6.038,148.371
C03587=1220.713,185.766,-55.334,-177.615,6.037,148.372
C03588=1220.717,185.496,-55.309,-177.617,6.036,148.372
C03589=1220.722,185.226,-55.284,-177.620,6.034,148.372
C03590=1220.728,184.956,-55.259,-177.623,6.032,148.373
C03591=1220.732,184.708,-55.237,-177.626,6.030,148.373
C03592=1220.737,184.459,-55.213,-177.628,6.029,148.374
C03593=1220.742,184.210,-55.190,-177.631,6.027,148.374
C03594=1220.746,183.961,-55.167,-177.633,6.026,148.374
C03595=1220.751,183.712,-55.144,-177.636,6.024,148.375
C03596=1220.755,183.464,-55.122,-177.639,6.022,148.375
C03597=1220.760,183.215,-55.099,-177.641,6.021,148.376
C03598=1220.765,182.965,-55.075,-177.644,6.020,148.376
C03599=1220.769,182.716,-55.053,-177.646,6.018,148.376
C03600=1220.774,182.468,-55.030,-177.649,6.016,148.377
C03601=1220.778,182.219,-55.008,-177.652,6.015,148.377
C03602=1220.783,181.969,-54.985,-177.654,6.013,148.378
C03603=1220.788,181.720,-54.962,-177.657,6.012,148.378
C03604=1220.792,181.472,-54.939,-177.659,6.011,148.378
C03605=1220.797,181.223,-54.916,-177.662,6.009,148.379
C03606=1220.801,180.974,-54.894,-177.665,6.007,148.379
C03607=1220.806,180.725,-54.870,-177.667,6.005,148.380
C03608=1220.811,180.476,-54.849,-177.669,6.004,148.380
C03609=1220.816,180.227,-54.825,-177.672,6.003,148.380
C03610=1220.820,179.979,-54.803,-177.675,6.001,148.381
C03611=1220.825,179.729,-54.780,-177.677,6.000,148.381
C03612=1220.829,179.481,-54.758,-177.680,5.998,148.382
C03613=1220.834,179.231,-54.735,-177.683,5.996,148.382
C03614=1220.838,178.983,-54.712,-177.685,5.995,148.382
C03615=1220.843,178.734,-54.689,-177.687,5.994,148.383
C03616=1220.848,178.485,-54.667,-177.691,5.992,148.383
C03617=1220.852,178.236,-54.644,-177.693,5.991,148.384
C03618=1220.857,177.987,-54.622,-177.695,5.989,148.384
C03619=1220.862,177.738,-54.599,-177.698,5.987,148.384
C03620=1220.866,177.489,-54.577,-177.700,5.986,148.385
C03621=1220.872,177.240,-54.554,-177.703,5.985,148.385
C03622=1220.876,176.991,-54.532,-177.706,5.983,148.386
C03623=1220.880,176.742,-54.509,-177.708,5.981,148.386
C03624=1220.885,176.493,-54.487,-177.711,5.980,148.387
C03625=1220.889,176.245,-54.464,-177.713,5.978,148.387
C03626=1220.894,175.995,-54.441,-177.716,5.977,148.387
C03627=1220.899,175.747,-54.419,-177.718,5.976,148.388
C03628=1220.903,175.498,-54.397,-177.721,5.974,148.388
C03629=1220.908,175.248,-54.374,-177.724,5.972,148.389
C03630=1220.913,175.000,-54.352,-177.726,5.972,148.389
C03631=1220.918,174.750,-54.329,-177.729,5.970,148.390
C03632=1220.922,174.502,-54.306,-177.732,5.968,148.390
C03633=1220.927,174.253,-54.285,-177.734,5.967,148.390
C03634=1220.932,174.003,-54.262,-177.736,5.965,148.391
C03635=1220.936,173.755,-54.240,-177.739,5.965,148.391
C03636=1220.940,173.506,-54.217,-177.742,5.963,148.392
C03637=1220.945,173.256,-54.195,-177.744,5.961,148.392
C03638=1220.950,173.008,-54.172,-177.746,5.960,148.392
C03639=1220.954,172.759,-54.150,-177.750,5.958,148.393
C03640=1220.960,172.510,-54.128,-177.752,5.957,148.393
C03641=1220.964,172.261,-54.105,-177.754,5.956,148.394
C03642=1220.968,172.012,-54.083,-177.757,5.954,148.394
C03643=1220.974,171.763,-54.061,-177.760,5.952,148.395
